MW_Float( WORD_STRONG:= MesBlock[1][1], 	WORD_WEAK := MesBlock[1][2],  VAR_OUT:=MesDataExd.MesData.MesI1);
MW_Float( WORD_STRONG:= MesBlock[1][3], 	WORD_WEAK := MesBlock[1][4],  VAR_OUT:=MesDataExd.MesData.MesI2);
MW_Float( WORD_STRONG:= MesBlock[1][5], 	WORD_WEAK := MesBlock[1][6],  VAR_OUT:=MesDataExd.MesData.MesI3);
MW_Float( WORD_STRONG:= MesBlock[1][7], 	WORD_WEAK := MesBlock[1][8],  VAR_OUT:=MesDataExd.MesData.MesI0);
MW_Float( WORD_STRONG:= MesBlock[1][15], 	WORD_WEAK := MesBlock[1][16], VAR_OUT:=MesDataExd.Thermal_Overload);
MW_Float( WORD_STRONG:= MesBlock[1][17], 	WORD_WEAK := MesBlock[1][18], VAR_OUT:=MesDataExd.MesData.MesFreq);


MesDataExd.Comut 			:= WORD_TO_BOOL(MesBlock[2][7]);
MesDataExd.CB_Close 		:= WORD_TO_BOOL(MesBlock[2][8]);
MesDataExd.CB_In_Alarm 		:= WORD_TO_BOOL(MesBlock[2][9]);
MesDataExd.Trip_Counter 	:= WORD_TO_INT(MesBlock[3][3]);

END_IF
END_METHOD

END_FUNCTION_BLOCK

// ---- 01_Equipement_Library/ProtectRelay/FB_ProtectRelay_REF615.TcPOU
FUNCTION_BLOCK FB_ProtectRelay_REF615 EXTENDS FB_ProtectRelay_Base
VAR_INPUT PERSISTENT
	{attribute 'OPC.UA.DA' := '1'} 
		ParamIPAddress				: STRING 	:= '192.168.20.66'; 	// (NA)Config: IP Adress of PV INverter
	{attribute 'OPC.UA.DA' := '1'} 
		ParamUnitID 				: BYTE  	:= 1; 			  		// (NA)   Modbus Unit ID. 
	{attribute 'OPC.UA.DA' := '1'} 
		ParamTCPPort				: UINT		:= 502;					// (NA) TCP port for modbus
		

//		ParamTempoComAlarm			: TIME 		:= T#2S;
//		ParamTempoComWarning		: TIME		:= T#2S;
		ParamNominalCurrent			: REAL 		:= 100 ; 				// (A) Nominal current set in the protection relay.
		
END_VAR

VAR
	// M_ALARMMANAGEMENT		
//		TON_ComAlarm				: TON;
//		TON_ComWarning				: TON;	
//		MesWarningCom				: BOOL;
//		MesAlarmCom					: BOOL;
	// M_READ VARIABLES//
		AX_ModbusRead		   		: ARRAY [1..3] OF FB_ModbusRead ; 					// (NA) FB for Modbus Reading
		                                        
		MesBlock_Temp 				: ARRAY [1..3] OF ARRAY[1..120]  OF WORD; 			// (NA) Temporary Block with multiple modbus reading (Caution : Double Word variables)

	MesDataExd		AT %Q* 	: ProtectRelay_REFIO ; 
	

	// M_STATEMANAGER//
	
END_VAR

METHOD M_AlarmManagement
//////////////////
// Manages IntelliGen Alarms
/////////////////

VAR 
	// Method local variables (reinitialized at each cycle) 
	FB_AlarmCodeManager : FB_AlarmCodeManager ; 

	KK					: BYTE;		// For Loop 
	
	ComWarning			: BOOL;		// Aggregated Wcommunication warning
	ComAlarm			: BOOL;		// Aggregated communication Alarm

	MesWarningCom: BOOL;
END_VAR

	//Alarm
	
	TON_ComAlarm	(IN:= (AX_ModbusRead[1].ModbusReadAlarm) AND (AX_ModbusRead[2].ModbusReadAlarm) AND (AX_ModbusRead[3].ModbusReadAlarm) , PT:= ParamTempoComAlarm, 	Q=> MesDataExd.MesData.MesAlarmCom) ;	
//	TON_ComWarning	(IN:= (AX_ModbusRead[1].ModbusReadAlarm) OR  (AX_ModbusRead[2].ModbusReadAlarm) OR  (AX_ModbusRead[3].ModbusReadAlarm) , PT:= ParamTempoComWarning, 	Q=>MesWarningCom) ;	

	MesWarningCom :=(AX_ModbusRead[1].ModbusReadAlarm) OR  (AX_ModbusRead[2].ModbusReadAlarm) OR  (AX_ModbusRead[3].ModbusReadAlarm) ; 


	
// ALARM CODE //
	FB_AlarmCodeManager(
		bAlarm1			:= MesDataExd.MesData.MesAlarmImax,  				//  Max I>>0  fault  
		bAlarm2			:= FALSE , 										//
		bAlarm3			:= MesDataExd.MesData.MesAlarmCom , 			// Communication alarm #COM
		bAlarm4			:= MesDataExd.MesData.MesAlarmTCS, 		        // Trip circuit Supervision alarm .     
		bAlarm5			:= FALSE, 										// 
		bAlarm6			:= FALSE, 										// 
		bAlarm7			:= False, 										// 
		bAlarm8			:= False, 										// 
		bAlarm9			:= FALSE, 										//
		bAlarm10		:= FALSE, 										//
		bAlarm11		:= FALSE,                       				//
		bAlarm12		:= FALSE,                       				//
		bAlarm13		:= FALSE, 										//
		bAlarm14		:= FALSE, 										// 
		bAlarm15		:= FALSE , 										// 
		wAlarmCode		=>MesDataExd.MesData.MesAlarmCode);

// WARNING CODE //
	FB_AlarmCodeManager(
 		bAlarm1			:= MesWarningCom,								// Bad communication	#COM			
		bAlarm2			:= FALSE ,										// 
		bAlarm3			:= FALSE , 										//		
		bAlarm4			:= FALSE, 						                //
		bAlarm5			:= FALSE, 						                //
		bAlarm6			:= FALSE, 						                //
		bAlarm7			:= FALSE,                                       //
		bAlarm8			:= FALSE,                                       //
		bAlarm9			:= FALSE,                                       //
		bAlarm10		:= FALSE,                                       //
		bAlarm11		:= FALSE,                                       //
		bAlarm12		:= FALSE,                                       //
		bAlarm13		:= FALSE,                                       //
		bAlarm14		:= FALSE,                                       //
		bAlarm15		:= FALSE,                                       //
		wAlarmCode		=>MesDataExd.MesData.MesWarningCode);	

// EVENT CODE //
	FB_AlarmCodeManager(
 		bAlarm1			:= FALSE,		//				
		bAlarm2			:= FALSE,	    //
		bAlarm3			:= FALSE,		//	
		bAlarm4			:= FALSE, 		//				
		bAlarm5			:= FALSE, 		//				
		bAlarm6			:= FALSE, 		//				
		bAlarm7			:= FALSE,       //
		bAlarm8			:= FALSE,       //
		bAlarm9			:= FALSE,       //
		bAlarm10		:= FALSE,       //
		bAlarm11		:= FALSE,       //
		bAlarm12		:= FALSE,       //
		bAlarm13		:= FALSE,       //
		bAlarm14		:= FALSE,       //
		bAlarm15		:= FALSE,       //
		wAlarmCode		=>MesDataExd.MesData.MesEventCode);
END_METHOD

METHOD M_Read
//////////////////
//  Read Modbus Variable for PCS . 
/////////////////
VAR 
	// Method local variables (reinitialized at each cycle) 
		
		AX_Addr				: ARRAY[1..3] OF UINT := [138, 		9409, 	171 ];
		AX_Qty				: ARRAY[1..3] OF UINT := [4, 		4, 	36	];
		
	
END_VAR
// CP-Read / Write 

MesDataExd.MesData.MesCP_Read := MesCP_Read ; 


// System BMS 
IF MesCP_Read  THEN	

AX_ModbusRead[1]
(
	pDestAddr 		:= ADR(MesBlock_Temp[1]),
	sIPAddr 		:= ParamIPAddress,
	tTimeout 		:= ParamTimeout,
	nQuantity 		:= AX_Qty[1],
	ntcpport 		:= ParamTCPPort,
	nMBAddr 		:= AX_Addr[1]-1,
	nUnitID 		:= ParamUnitID,
	cbLength 		:= SIZEOF(MesBlock_Temp[1]),
	ClockRead 		:= ClockRead AND MesCP_Read,
	Reset 			:= CmdClearFault_G OR IN_CmdReset_L,
);

AX_ModbusRead[2]
(
	pDestAddr 		:= ADR(MesBlock_Temp[2]),
	sIPAddr 		:= ParamIPAddress,
	tTimeout 		:= ParamTimeout,
	nQuantity 		:= AX_Qty[2],
	ntcpport 		:= ParamTCPPort,
	nMBAddr 		:= AX_Addr[2]-1,
	nUnitID 		:= ParamUnitID,
	cbLength 		:= SIZEOF(MesBlock_Temp[2]),
	ClockRead 		:= ClockRead AND MesCP_Read,
	Reset 			:= CmdClearFault_G OR IN_CmdReset_L
);

AX_ModbusRead[3]
(
	pDestAddr 		:= ADR(MesBlock_Temp[3]),
	sIPAddr 		:= ParamIPAddress,
	tTimeout 		:= ParamTimeout,
	nQuantity 		:= AX_Qty[3],
	ntcpport 		:= ParamTCPPort,
	nMBAddr 		:= AX_Addr[3]-1,
	nUnitID 		:= ParamUnitID,
	cbLength 		:= SIZEOF(MesBlock_Temp[3]),
	ClockRead 		:= ClockRead AND MesCP_Read,
	Reset 			:= CmdClearFault_G OR IN_CmdReset_L
);



	


MesDataExd.MesData.MesI1 	:= WORD_TO_REAL(MesBlock_Temp[1][1])/1000*ParamNominalCurrent;
MesDataExd.MesData.MesI2 	:= WORD_TO_REAL(MesBlock_Temp[1][2])/1000*ParamNominalCurrent;
MesDataExd.MesData.MesI3 	:= WORD_TO_REAL(MesBlock_Temp[1][3])/1000*ParamNominalCurrent;
MesDataExd.MesData.MesI0 	:= WORD_TO_REAL(MesBlock_Temp[1][4])/1000*ParamNominalCurrent;


MesDataExd.MesData.MesImax1	:= WORD_TO_REAL(MesBlock_Temp[2][1])/1000*ParamNominalCurrent;
MesDataExd.MesData.MesImax2	:= WORD_TO_REAL(MesBlock_Temp[2][2])/1000*ParamNominalCurrent;
MesDataExd.MesData.MesImax3	:= WORD_TO_REAL(MesBlock_Temp[2][3])/1000*ParamNominalCurrent;
MesDataExd.MesData.MesImax0	:= WORD_TO_REAL(MesBlock_Temp[2][4])/1000*ParamNominalCurrent;


MesDataExd.MesTransfoAlarm		:= MesBlock_Temp[3][31].0 ;
MesDataExd.MesSWOpened			:= MesBlock_Temp[3][31].4 ;
MesDataExd.MesSWClosed			:= MesBlock_Temp[3][31].6 ;
MesDataExd.MesEarth				:= MesBlock_Temp[3][31].8 ;
MesDataExd.MesSF6Low			:= MesBlock_Temp[3][31].10;
MesDataExd.MesSF6Unsufficient	:= MesBlock_Temp[3][31].12;
MesDataExd.MesTransfoWarning		:= MesBlock_Temp[3][31].14;

MesDataExd.MesClosed	        := MesBlock_Temp[3][30].2;
MesDataExd.MesOpened	        := MesBlock_Temp[3][30].4;
MesDataExd.MesComutLocal				:= NOT MesBlock_Temp[3][30].6;

MesDataExd.MesData.MesAlarmImax				:= MesBlock_Temp[3][3].1 ; // Max I ou Max I Inverse. Maintenu jusque l'acquittement.  
//MesDataExd.MesData.MesAlarmTCS				:=  ; 

END_IF

//MesDataExd.MesData.MesAlarmUminrmUmin	:= ; 

// Properties update
MesDataExd.MesData.MesI := (MesDataExd.MesData.MesI1 + MesDataExd.MesData.MesI2 + MesDataExd.MesData.MesI3)/3 ;
END_METHOD

END_FUNCTION_BLOCK

// ---- 01_Equipement_Library/ProtectRelay/FB_ProtectRelay_SepamT20.TcPOU
FUNCTION_BLOCK FB_ProtectRelay_SepamT20 EXTENDS FB_ProtectRelay_Base
//////////////////
// SEPAM system for High Voltage or Low Voltage Grid Protection . 
//////////////////
VAR_INPUT PERSISTENT
	// Parameters of the Object (instance/model specific) 
	 
END_VAR

VAR_OUTPUT
	//Child objects
	OutFBCompleteted						: BOOL;
END_VAR

VAR_INPUT
	InUnitID            : DINT;			// (NA)   ID FOR SEPAM T20 Modbus Unit ID. 

	// I/O Inputs		
END_VAR

VAR
	//M_Read
	FB_ModbusRead_I1						: FB_ReadModbusRTU_V2; 				// (NA) FB for Modbus Reading
	FB_ModbusRead_I2						: FB_ReadModbusRTU_V2; 				// (NA) FB for Modbus Reading
	FB_ModbusRead_I3						: FB_ReadModbusRTU_V2; 				// (NA) FB for Modbus Reading
	ParamTimeoutRTU							: TIME:=T#10S;
	MesBlock1_Temp							: ARRAY [0..36] OF WORD;
	MesBlock2_Temp							: WORD;
	MesBlock3_Temp							: WORD;
	MesModbusAlarmCode						: UDINT;							// (NA) Modbus Read Alarm Code
	MesModbusAlarmCode2						: UDINT;							// (NA) Modbus Read Alarm Code
	MesModbusAlarmCode3						: UDINT;							// (NA) Modbus Read Alarm Code
	ModbusReadAlarm 						: BOOL;								// (NA) Modbus Read Alarm for communications
	ModbusReadAlarm2 						: BOOL;	
	ModbusReadAlarm3 						: BOOL;	
	AX_bRead 								: ARRAY [1..3] OF BOOL;
	CalAllCompleted							: BOOL;
	//M_ALARMMANAGEMENT VARIABLES//

	//M_Execute
	AllNotBusy								: BOOL;
	TP_Read									: TP;
	RTrig									: R_TRIG;
//	ClockRead								: BOOL;
	
	//EValuate//
MesDataExd					AT %Q* 		: ProtectRelay_T20;
	

		
END_VAR

METHOD M_AlarmManagement
//////////////////
// Manages Sepam Alarms. Alarms opens HT CB until Sepam manual Reset . Warning Opens CB-L but does not maintain warning
/////////////////

VAR 
	// Method local variables (reinitialized at each cycle) 
	FB_AlarmCodeManager 	: FB_AlarmCodeManager ; 
 	ComWarning				: BOOL;
	ComAlarms				: BOOL;
END_VAR
ComWarning	:= ModbusReadAlarm OR ModbusReadAlarm2 OR ModbusReadAlarm3;
ComAlarms	:= ModbusReadAlarm OR ModbusReadAlarm2 OR ModbusReadAlarm3;

// ALARM CODE //
	FB_AlarmCodeManager(
		bAlarm1				:= FALSE,									//	
		bAlarm2				:= MesDataExd.MesGlobalWarming > 95 ,		// Calc of Warming TR from Sepam > 95 % OF T° Max				
		bAlarm3				:= ComAlarms ,								// Communication alarm  #COM
		bAlarm4				:= FALSE,     							//
		bAlarm5				:= FALSE,         						// 
		bAlarm6				:= FALSE, 								// 
		bAlarm7				:= FALSE, //
		bAlarm8				:= FALSE, //
		bAlarm9				:= FALSE, //
		bAlarm10			:= FALSE, //
		bAlarm11			:= FALSE, //
		bAlarm12			:= FALSE, //
		bAlarm13			:= FALSE, //
		bAlarm14			:= FALSE, //
		bAlarm15			:= FALSE , 	// 
		wAlarmCode			=>MesDataExd.MesData.MesAlarmCode);

// WARNING CODE //
	FB_AlarmCodeManager(
		bAlarm1			:= ComWarning, 							//  At least One Register do not responce #COM
		bAlarm2			:= FALSE,//  MesDataExd.MesData.MesPartialdefault, 			// Sepam in partial defaut IO, Tor fault
		bAlarm4			:= MesDataExd.MesGlobalWarming > 80, 	// Calc of Warming TR from Sepam > 80 % OF T° Max
		bAlarm5			:= FALSE, //
		bAlarm6			:= FALSE, //
		bAlarm7			:= FALSE, //
		bAlarm8			:= FALSE, //
		bAlarm9			:= FALSE, //
		bAlarm10		:= FALSE, //
		bAlarm11		:= FALSE, //
		bAlarm12		:= FALSE, //
		bAlarm13		:= FALSE, //
		bAlarm14		:= FALSE, //
		bAlarm15		:= FALSE, //
		wAlarmCode		=>MesDataExd.MesData.MesWarningCode);

// EVENT CODE //
	FB_AlarmCodeManager(
		bAlarm1			:=FALSE, 		// 
		bAlarm2			:=FALSE, 		// 
		bAlarm3			:=FALSE, 		// 
		bAlarm4			:=FALSE, 		// 
		bAlarm5			:=FALSE, 
		bAlarm6			:=FALSE, 
		bAlarm7			:=FALSE, 
		bAlarm8			:=FALSE, 
		bAlarm9			:=FALSE, 
		bAlarm10		:=FALSE, 
		bAlarm11		:=FALSE, 
		bAlarm12		:=FALSE, 
		bAlarm13		:=FALSE, 
		bAlarm14		:=FALSE, 
		bAlarm15		:=FALSE, 
		wAlarmCode		=>MesDataExd.MesData.MesEventCode);
END_METHOD

METHOD M_Init
VAR_INPUT
END_VAR
OutFBCompleteted := FALSE;
TP_Read(PT := ParamClockReadTime);
FB_ModbusRead_I1(InTimeout:= ParamTimeoutRTU,
				 InUnitID:= DINT_TO_BYTE(InUnitID),
				 InQuantity:= 36,	
				 InFunctionRead := 1);
				 
FB_ModbusRead_I2(InTimeout:= ParamTimeoutRTU,
				 InUnitID:= DINT_TO_BYTE(InUnitID),
				 InQuantity:= 1,	
				 InFunctionRead := 1);

				 
FB_ModbusRead_I3(InTimeout:= ParamTimeoutRTU,
				 InUnitID:= DINT_TO_BYTE(InUnitID),
				 InQuantity:= 1,	
				 InFunctionRead := 1);
END_METHOD

METHOD M_Read
//////////////////
//  Method Calls 
/////////////////

VAR 
//local variables (reinitialized at each cycle) 
	Busy1 : BOOL;
	Error1: BOOL;
	Busy2 : BOOL;
	Error2: BOOL;
	Busy3 : BOOL;
	Error3: BOOL;
	MW 					: FB_MergeWordsToDint; 
END_VAR
// CP-Read / Write 

MesDataExd.MesData.MesCP_Read := MesCP_Read ; 

IF MesCP_Read  THEN	



AllNotBusy:=TRUE;
AllNotBusy:=NOT(FB_ModbusRead_I1.OutBusy) AND NOT(FB_ModbusRead_I2.OutBusy) AND NOT(FB_ModbusRead_I3.OutBusy) AND AllNotBusy;



OutFBCompleteted:=FALSE;

// MODBUS REQUEST//
	//First register
		FB_ModbusRead_I1(InClockRead:= ClockRead,				
						InStartAddr:= 16#106,
						InAddrDest := ADR(MesBlock1_Temp),
						OutBusy => Busy1,
						OutErrorMbRead => Error1, 
						OutErrorId => MesModbusAlarmCode
						   );
						
		IF FB_ModbusRead_I1.OutbCompleted THEN
			ModbusReadAlarm := Error1;
			AX_bRead[1] 		:= TRUE;
		ELSIF NOT busy1 AND Error1 THEN
			ModbusReadAlarm := Error1;
		END_IF
	//Seconde Register
		FB_ModbusRead_I2(InClockRead:= ClockRead,				
						InStartAddr:= 16#1004,
						InAddrDest := ADR(MesBlock2_Temp),
						OutBusy => Busy2,
						OutErrorMbRead => Error2, 
						OutErrorId => MesModbusAlarmCode2
						   );		
		IF FB_ModbusRead_I2.OutbCompleted THEN
			ModbusReadAlarm2 := Error2;
			AX_bRead[2] 		:= TRUE;
		ELSIF NOT busy1 AND Error1 THEN
			ModbusReadAlarm2 := Error2;
		END_IF
	
	
	
	//Third Register
		FB_ModbusRead_I3(InClockRead:= ClockRead,				
						InStartAddr:= 16#1007,
						InAddrDest := ADR(MesBlock3_Temp),
						OutBusy => Busy3,
						OutErrorMbRead => Error3, 
						OutErrorId => MesModbusAlarmCode3
						   );		
		IF FB_ModbusRead_I3.OutbCompleted THEN
			ModbusReadAlarm3 := Error3;
			AX_bRead[3] 		:= TRUE;
		ELSIF NOT busy3 AND Error3 THEN
			ModbusReadAlarm3 := Error3;
		END_IF
	
	
CalAllCompleted :=  AX_bRead[1] AND AX_bRead[2] AND AX_bRead[3];
OutFBCompleteted := CalAllCompleted;	

//CHECK IF ALL MODBUS REQUESTS ARE FINISHED
	IF (CalAllCompleted) THEN
//RESETING CLOCK READ FOR EACH REQUEST
		AX_bRead[1]:= FALSE;
		AX_bRead[2]:= FALSE;
		AX_bRead[3]:= FALSE;
		CalAllCompleted := FALSE;
	END_IF
	
MW( WORD_STRONG:= MesBlock1_Temp[0], SIGNED:=FALSE, FIX:=0 , SIZE:=1, VAR_OUT 	:=MesDataExd.MesData.MesI1);
MW( WORD_STRONG:= MesBlock1_Temp[1], SIGNED:=FALSE, FIX:=0 , SIZE:=1, VAR_OUT 	:=MesDataExd.MesData.MesI2);
MW( WORD_STRONG:= MesBlock1_Temp[2], SIGNED:=FALSE, FIX:=0 , SIZE:=1, VAR_OUT 	:=MesDataExd.MesData.MesI3);
MW( WORD_STRONG:= MesBlock1_Temp[33], SIGNED:=FALSE, FIX:=2 , SIZE:=1, VAR_OUT	:=MesDataExd.MesData.MesFreq);
MW( WORD_STRONG:= MesBlock1_Temp[34], SIGNED:=TRUE, FIX:=0 , SIZE:=1, VAR_OUT 	:=MesDataExd.MesP);
MW( WORD_STRONG:= MesBlock1_Temp[35], SIGNED:=TRUE, FIX:=0 , SIZE:=1, VAR_OUT 	:=MesDataExd.MesQ);
MW( WORD_STRONG:= MesBlock1_Temp[36], SIGNED:=TRUE, FIX:=0 , SIZE:=1, VAR_OUT 	:=MesDataExd.MesS);
MW( WORD_STRONG:= MesBlock2_Temp, SIGNED:=FALSE, FIX:=-1 , SIZE:=1, VAR_OUT 	:=MesDataExd.MesTripProtec);
MW( WORD_STRONG:= MesBlock3_Temp, SIGNED:=FALSE, FIX:=0 , SIZE:=1, VAR_OUT 		:=MesDataExd.MesGlobalWarming);

END_IF
END_METHOD

END_FUNCTION_BLOCK

// ---- 01_Equipement_Library/ProtectRelay/FB_ProtectRelay_VIP410.TcPOU
FUNCTION_BLOCK FB_ProtectRelay_VIP410 EXTENDS FB_ProtectRelay_Base
//////////////////
// SEPAM system for High Voltage or Low Voltage Grid Protection . 
//////////////////
VAR_INPUT PERSISTENT
	{attribute 'OPC.UA.DA' := '1'} 
	ParamTcpPort				: UINT:=502;		(* (NA) Tcp port *)
	{attribute 'OPC.UA.DA' := '1'} 
	ParamIPAddress				: STRING;       	(* (NA) IP address*)
	{attribute 'OPC.UA.DA' := '1'} 
	ParamUnitID					: BYTE;         	(* (NA) Unit ID*)
	{attribute 'OPC.UA.DA' := '1'}
	ParamClockInputTime 		: TIME:= TIME#5S;   (* (Time) Read Modbus Frequency*)
END_VAR

VAR_OUTPUT
	
END_VAR

VAR_INPUT
	IN_MesTrip_IO				: BOOL ; 
END_VAR

VAR
	
	MesDataExd		AT %Q* 		: ProtectRelay_VIP410;
	FB_ModbusRead	          	: ARRAY[1..4] OF FB_ModbusRead; 
	ClockReadInput				: BOOL;

	MesBlock1_Temp 				: ARRAY [1..1] OF WORD ; 
	MesBlock2_Temp 				: ARRAY [1..20] OF WORD ; 
	MesBlock3_Temp 				: ARRAY [1..8] OF WORD ; 
	MesBlock4_Temp 				: ARRAY [1..2] OF WORD ; 
	AX_ModbusReadAlarm			: ARRAY[1..4] OF BOOL;
	AX_ModbusReadAlarmId		: ARRAY[1..4] OF UDINT;	
END_VAR

METHOD M_AlarmManagement
//////////////////
// Manages Sepam Alarms. Alarms opens HT CB until Sepam manual Reset . Warning Opens CB-L but does not maintain warning
/////////////////

VAR 
	// Method local variables (reinitialized at each cycle) 
	FB_AlarmCodeManager 	: FB_AlarmCodeManager ; 
	RS_Trip					: SR;
	ComWarning: BOOL ;
END_VAR
RS_Trip(SET1 := IN_MesTrip_IO  , Reset := CmdClearFault_G OR IN_CmdReset_L ); // SR FB for keep fire if burn .

TON_ComAlarm(IN:= AX_ModbusReadAlarm[1] AND AX_ModbusReadAlarm[2] AND AX_ModbusReadAlarm[3] AND AX_ModbusReadAlarm[4] , PT:= ParamTempoComAlarm, Q=>MesdataExd.MesData.MesAlarmCom) ;	

ComWarning := AX_ModbusReadAlarm[1] OR AX_ModbusReadAlarm[2] OR AX_ModbusReadAlarm[3] OR AX_ModbusReadAlarm[4] ; 

// ALARM CODE //
	FB_AlarmCodeManager(
		bAlarm1				:= RS_Trip.Q1,							// General trip
		bAlarm2				:= NOT IN_MesWatchDog_IO,				// Watchdog lost
		bAlarm3				:= MesdataExd.MesData.MesAlarmCom,		// Communication Alarm
		bAlarm4				:= FALSE,     							// 
		bAlarm5				:= FALSE,         						// 
		bAlarm6				:= FALSE, 								// 
		bAlarm7				:= FALSE, 								// 
		bAlarm8				:= FALSE, 								// 
		bAlarm9				:= FALSE, 								// 
		bAlarm10			:= FALSE, 								// 
		bAlarm11			:= FALSE, 								// 
		bAlarm12			:= FALSE, 								// 
		bAlarm13			:= FALSE, 								// 
		bAlarm14			:= FALSE, 								// 
		bAlarm15			:= FALSE,								//  	
		wAlarmCode			=> MesdataExd.MesData.MesAlarmCode);

// WARNING CODE //
	FB_AlarmCodeManager(
		bAlarm1			:= FALSE,									// 
		bAlarm2			:= FALSE,									// 
		bAlarm4			:= FALSE,									// 
		bAlarm5			:= FALSE,									// 
		bAlarm6			:= FALSE,									// 
		bAlarm7			:= FALSE,									//  
		bAlarm8			:= FALSE,									// 
		bAlarm9			:= FALSE,									// 
		bAlarm10		:= FALSE,									// 
		bAlarm11		:= FALSE,									// 
		bAlarm12		:= FALSE,									// 
		bAlarm13		:= FALSE,									// 
		bAlarm14		:= FALSE,									//
		bAlarm15		:= FALSE,									//
		wAlarmCode		=> MesdataExd.MesData.MesWarningCode);

// EVENT CODE //
	FB_AlarmCodeManager(
		bAlarm1			:=FALSE, 									// 
		bAlarm2			:=FALSE, 									// 
		bAlarm3			:=FALSE, 									// 
		bAlarm4			:=FALSE, 									// 
		bAlarm5			:=FALSE, 									// 
		bAlarm6			:=FALSE, 									// 
		bAlarm7			:=FALSE, 									// 
		bAlarm8			:=FALSE, 									// 
		bAlarm9			:=FALSE, 									// 
		bAlarm10		:=FALSE, 									// 
		bAlarm11		:=FALSE, 									// 
		bAlarm12		:=FALSE, 									// 
		bAlarm13		:=FALSE, 									// 
		bAlarm14		:=FALSE, 									//
		bAlarm15		:=FALSE, 									//
		wAlarmCode		=> MesdataExd.MesData.MesEventCode);
END_METHOD

METHOD M_Evaluate
VAR_INPUT
END_VAR

VAR
END_VAR

// Structure update 
	MesDataExd.MesData.MesI		:= (MesDataExd.MesData.MesI1 + MesDataExd.MesData.MesI2 + MesDataExd.MesData.MesI3 )/3 ; 
	///MesDataExd.MesData	:= MesData;
END_METHOD

METHOD M_Init
VAR_INPUT
END_VAR
END_METHOD

METHOD M_Read
//////////////////
//  Method Calls 
/////////////////

VAR_INPUT
	
END_VAR
VAR 
	MW					: FB_MergeWordsToFloat;
END_VAR
// CP-Read / Write 

MesDataExd.MesData.MesCP_Read := MesCP_Read ; 

IF MesCP_Read  THEN	



FB_ModbusRead[1]
	(
		nTCPPort		:= ParamTcpPort,
		ClockRead		:= MesCP_Read AND ClockRead	, 
		Reset			:= CmdClearFault_G OR IN_CmdReset_L,
		sIPAddr			:= ParamIPAddress ,
		nUnitID			:= ParamUnitID, 
		tTimeout		:= T#5S,
		nQuantity		:= 1, 
		nMBAddr			:= 40000 , 
		cbLength		:= SIZEOF(MesBlock1_Temp) , 
		pDestAddr		:= ADR(MesBlock1_Temp) , 
		ModbusReadAlarm	=> AX_ModbusReadAlarm[1] , 
		ErrorId			=> AX_ModbusReadAlarmId[1]
	);
	
FB_ModbusRead[2]
	(
		nTCPPort		:= ParamTcpPort,
		ClockRead		:= MesCP_Read AND ClockRead	, 
		Reset			:= CmdClearFault_G OR IN_CmdReset_L,
		sIPAddr			:= ParamIPAddress ,
		nUnitID			:= ParamUnitID, 
		tTimeout		:= T#5S,
		nQuantity		:= 20, 
		nMBAddr			:= 40200 , 
		cbLength		:= SIZEOF(MesBlock2_Temp) , 
		pDestAddr		:= ADR(MesBlock2_Temp) , 
		ModbusReadAlarm	=> AX_ModbusReadAlarm[2], 
		ErrorId			=> AX_ModbusReadAlarmId[2]
	);

FB_ModbusRead[3]
	(
		nTCPPort		:= ParamTcpPort,
		ClockRead		:= MesCP_Read AND ClockRead	, 
		Reset			:= CmdClearFault_G OR IN_CmdReset_L,
		sIPAddr			:= ParamIPAddress ,
		nUnitID			:= ParamUnitID, 
		tTimeout		:= T#5S,
		nQuantity		:= 8, 
		nMBAddr			:= 40254 , 
		cbLength		:= SIZEOF(MesBlock3_Temp) , 
		pDestAddr		:= ADR(MesBlock3_Temp) , 
		ModbusReadAlarm	=> AX_ModbusReadAlarm[3], 
		ErrorId			=> AX_ModbusReadAlarmId[3]
	);
	
FB_ModbusRead[4]
	(
		nTCPPort		:= ParamTcpPort,
		ClockRead		:= MesCP_Read AND ClockRead	, 
		Reset			:= CmdClearFault_G OR IN_CmdReset_L,
		sIPAddr			:= ParamIPAddress ,
		nUnitID			:= ParamUnitID, 
		tTimeout		:= T#5S,
		nQuantity		:= 2, 
		nMBAddr			:= 40351 , 
		cbLength		:= SIZEOF(MesBlock4_Temp) , 
		pDestAddr		:= ADR(MesBlock4_Temp) , 
		ModbusReadAlarm	=> AX_ModbusReadAlarm[4], 
		ErrorId			=> AX_ModbusReadAlarmId[4]
	);
	
	//COM
	MesdataExd.MesStatCom := WORD_TO_BOOL(MesBlock1_Temp[1]);
	//I
	MW( WORD_STRONG:= MesBlock2_Temp[2  ],	WORD_WEAK := MesBlock2_Temp[1  ], VAR_OUT := MesDataExd.MesData.MesI1 );		
	MW( WORD_STRONG:= MesBlock2_Temp[4  ],	WORD_WEAK := MesBlock2_Temp[3  ], VAR_OUT := MesDataExd.MesData.MesI2 );	
	MW( WORD_STRONG:= MesBlock2_Temp[6  ],	WORD_WEAK := MesBlock2_Temp[5  ], VAR_OUT := MesDataExd.MesData.MesI3 );
	MW( WORD_STRONG:= MesBlock2_Temp[8  ],	WORD_WEAK := MesBlock2_Temp[7  ], VAR_OUT := MesDataExd.MesData.MesI0 );	
	
	//AvgI
	MW( WORD_STRONG:= MesBlock2_Temp[10  ],	WORD_WEAK := MesBlock2_Temp[9  ], VAR_OUT 	:= MesDataExd.MesAvgI1 );	
	MW( WORD_STRONG:= MesBlock2_Temp[12  ],	WORD_WEAK := MesBlock2_Temp[11  ], VAR_OUT 	:= MesDataExd.MesAvgI2 );	
	MW( WORD_STRONG:= MesBlock2_Temp[14  ],	WORD_WEAK := MesBlock2_Temp[13  ], VAR_OUT 	:= MesDataExd.MesAvgI3 );	
	//Imax
	MW( WORD_STRONG:= MesBlock2_Temp[16  ],	WORD_WEAK := MesBlock2_Temp[15 ], VAR_OUT  := MesDataExd.MesData.MesImax1 );	
	MW( WORD_STRONG:= MesBlock2_Temp[18  ],	WORD_WEAK := MesBlock2_Temp[17  ], VAR_OUT := MesDataExd.MesData.MesImax2 );	
	MW( WORD_STRONG:= MesBlock2_Temp[20  ],	WORD_WEAK := MesBlock2_Temp[19  ], VAR_OUT := MesDataExd.MesData.MesImax3 );	

	//Itrip
	MW( WORD_STRONG:= MesBlock3_Temp[2  ],	WORD_WEAK := MesBlock3_Temp[1  ], VAR_OUT := MesDataExd.MesData.MesImax1 );		
	MW( WORD_STRONG:= MesBlock3_Temp[4  ],	WORD_WEAK := MesBlock3_Temp[3  ], VAR_OUT := MesDataExd.MesData.MesImax2 );	
	MW( WORD_STRONG:= MesBlock3_Temp[6  ],	WORD_WEAK := MesBlock3_Temp[5  ], VAR_OUT := MesDataExd.MesData.MesImax3 );
	MW( WORD_STRONG:= MesBlock3_Temp[8  ],	WORD_WEAK := MesBlock3_Temp[7  ], VAR_OUT := MesDataExd.MesI0Fault );	

	MesdataExd.ControlWord 	:= MesBlock4_Temp[1];
	MesdataExd.StatusWord 	:= MesBlock4_Temp[2];
	
END_IF
END_METHOD

END_FUNCTION_BLOCK

// ---- 01_Equipement_Library/ProtectRelay/FB_ProtectRelay_WIP1.TcPOU
FUNCTION_BLOCK FB_ProtectRelay_WIP1 EXTENDS FB_ProtectRelay_Base
VAR_INPUT
						
	
	

END_VAR

VAR_INPUT
	// I/O Inputs 		                                     				
		IN_MesAlarmImax_IO		: BOOL ; // IO max I  fault
		IN_MesAlarmUmin_IO		: BOOL ;  // IO Min U  Fault 
		
END_VAR


VAR
// M_ALARMMNGMT VARIABLES //
                            		
	CmdResetHVCell				: BOOL ; 
	// M_READ VARIABLES//
	
MesDataExd 		    AT %Q*  	: ProtectRelay_WIP1; 	
		


END_VAR

METHOD M_AlarmManagement
VAR 
	// Method local variables (reinitialized at each cycle) 
	FB_AlarmCodeManager : FB_AlarmCodeManager ; 

	ComWarning: BOOL;
	ComAlarm: BOOL;
	KK: BYTE;
	
END_VAR
// Detection Variables

MesDataExd.MesData.MesAlarmImax	:= IN_MesAlarmImax_IO ; 
MesDataExd.MesData.MesAlarmUmin :=  IN_MesAlarmUmin_IO ; 


// ALARM CODE //
	FB_AlarmCodeManager(
		bAlarm1	 := MesDataExd.MesData.MesAlarmImax,// Max I Fault 
		bAlarm2	 := MesDataExd.MesData.MesAlarmUmin,// Min U  Fault
		bAlarm3	 := FALSE, //
		bAlarm4	 := FALSE,//
		bAlarm5	 := FALSE, //
		bAlarm6	 := FALSE,//
		bAlarm7	 := FALSE, //
		bAlarm8	 := FALSE,//
		bAlarm9	 := FALSE, //
		bAlarm10 := FALSE,//
		bAlarm11 := FALSE, //
		bAlarm12 := FALSE,//
		bAlarm13 := FALSE, //
		bAlarm14 := FALSE,//														   
		bAlarm15 := FALSE,//									                      
		wAlarmCode	=>MesDataExd.MesData.MesAlarmCode);


// WARNING CODE //
	FB_AlarmCodeManager(
 		bAlarm1			:= FALSE, //
		bAlarm2			:= FALSE,//
        bAlarm3			:= FALSE, //
		bAlarm4			:= FALSE,// 
		bAlarm5			:= FALSE, // 
		bAlarm6			:= FALSE,// 
		bAlarm7			:= FALSE, // 
		bAlarm8			:= FALSE,// 
		bAlarm9			:= FALSE, // 
		bAlarm10		:= FALSE,// 
		bAlarm11		:= FALSE, // 
		bAlarm12		:= FALSE,//		 
		bAlarm13		:= FALSE,//		 
		bAlarm14		:= FALSE,  //
		bAlarm15		:= FALSE, //
		wAlarmCode	=>MesDataExd.MesData.MesWarningCode);
END_METHOD

METHOD M_Execute

// INITIALIZE // 
	IF bInit THEN
		M_Init() ; 
		bInit		:= FALSE ; 
		
	ELSIF IN_CmdReset_L THEN 
		bInit		:= TRUE ;
		
	END_IF





M_AlarmManagement() ;
END_METHOD

END_FUNCTION_BLOCK

// ---- 01_Equipement_Library/ProtectRelay/FB_ProtectRelay_SEPAM10a.TcPOU
FUNCTION_BLOCK FB_ProtectRelay_SEPAM10a EXTENDS FB_ProtectRelay_Base
VAR_INPUT
	InUnitID            : DINT;			// (NA)   SMA Modbus Unit ID. 
	
END_VAR
VAR_OUTPUT
	OutFBCompleteted   : BOOL;
	
END_VAR
VAR
// M_ALARMMNGMT VARIABLES //
		MesAlarmCode				: WORD ;  			// (NA) [P,H,B]   Alarm Word . 0: Synthesis , 1:SMA general alarm , 2:Communication Alarm , 3:, 4:, 5:, 6:, 7:, 8:, 9:, 10:, 11:, 12:, 13:, 14:, 15:, 16:
		MesWarningCode				: WORD ;  			// (NA) [P,H,B]   Warning Word . 0: Synthesis , 1:SMA general warning  , 2: , 3: , 4:, 5:, 6:, 7:, 8:, 9:, 10:, 11:, 12:, 13:, 14:, 15:, 16:		
  		MesEventCode				: WORD; 			// (NA) [P,H,B] Event Code. Acknowledgable.
                                              		

		MesComError					: BOOL ; 			// (NA) [P,H]  True if lost of communication
		MesAlarmCom					: BOOL ; 			// (NA) All modbus trame fail 
		
	// M_READ VARIABLES//
		FB_ModbusRead_I1          	: FB_ReadModbusRTU_V2; 				// (NA) FB for Modbus Reading
		MesDataExd		      	AT %Q* 	: ProtectRelay_S48; 	
		MesBlock1_Temp 				: ARRAY[0..7]  OF WORD; 			// (NA) Temporary Block with multiple modbus reading (Caution : Double Word variables)
		AX_bRead 					: ARRAY[1..2]  OF BOOL;
		ModbusReadAlarm             : BOOL;				// (NA) Modbus Read Alarm for communications
		MesModbusAlarmCode			: UDINT;							// (NA) Modbus Read Alarm Code
		CalAllCompleted				: BOOL;								// (NA) Returns the status of all modbus requests
	
		AllNotBusy					: BOOL:=TRUE;
		TP_Read						: LTP; 								// (NA) Tempo to define Modbus Reading Frequency
	//	ClockRead					: BOOL;								// (NA) Modbus reading Clock
		RTrig						: R_TRIG;
END_VAR

VAR CONSTANT
	    CstClockReadTime 		: LTIME := LTIME#1S;	  				// (Time) Read Modbus Frequency .	
END_VAR

METHOD M_AlarmManagement
VAR 
	// Method local variables (reinitialized at each cycle) 
	FB_AlarmCodeManager : FB_AlarmCodeManager ; 

	ComWarning: BOOL;
	ComAlarm: BOOL;
	KK: BYTE;
	
END_VAR
// Detection Variables
ComWarning 	:= ComWarning OR ModbusReadAlarm ; // At least one modbus trame did not work
ComAlarm	:= ComAlarm AND ModbusReadAlarm;  // All modbus trame did not work

MesComError := ComWarning ;  
MesAlarmCom := ComAlarm ;

// ALARM CODE //
	FB_AlarmCodeManager(
		bAlarm1	 := FALSE,//
		bAlarm2	 := FALSE,//
		bAlarm3	 := FALSE, 
		bAlarm4	 := FALSE,
		bAlarm5	 := FALSE,
		bAlarm6	 := FALSE,
		bAlarm7	 := FALSE,
		bAlarm8	 := FALSE,
		bAlarm9	 := FALSE,
		bAlarm10 := FALSE,
		bAlarm11 := FALSE,
		bAlarm12 := FALSE,
		bAlarm13 := FALSE,
		bAlarm14 := FALSE,														   
		bAlarm15 := FALSE,									                      
		wAlarmCode	=> MesAlarmCode);


// WARNING CODE //
	FB_AlarmCodeManager(
 		bAlarm1			:= FALSE,
		bAlarm2			:= FALSE,
        bAlarm3			:= FALSE,
		bAlarm4			:= FALSE, 
		bAlarm5			:= FALSE, 
		bAlarm6			:= FALSE, 
		bAlarm7			:= FALSE, 
		bAlarm8			:= FALSE, 
		bAlarm9			:= FALSE, 
		bAlarm10		:= FALSE, 
		bAlarm11		:= FALSE, 
		bAlarm12		:= FALSE, 
		bAlarm13		:= FALSE, 
		bAlarm14		:= FALSE, 
		bAlarm15		:= FALSE, 
		wAlarmCode	=> MesWarningCode);	
		
		
// EVENT CODE //
	FB_AlarmCodeManager(
		bAlarm1			:= FALSE,
		bAlarm2			:= FALSE,
		bAlarm3			:= FALSE,
		bAlarm4			:= FALSE, 		
		bAlarm5			:= FALSE, 
		bAlarm6			:= FALSE, 
		bAlarm7			:= FALSE, 
		bAlarm8			:= FALSE, 
		bAlarm9			:= FALSE, 
		bAlarm10		:= FALSE, 
		bAlarm11		:= FALSE, 
		bAlarm12		:= FALSE, 
		bAlarm13		:= FALSE, 
		bAlarm14		:= FALSE, 
		bAlarm15		:= FALSE, 
		wAlarmCode		=> MesEventCode);
END_METHOD

METHOD M_Execute
// INITIALIZE //
	IF NOT(bInit) THEN
		THIS^.M_Init();
		bInit := TRUE;
		
	END_IF
	IF bInit THEN
		AllNotBusy:=TRUE;
		AllNotBusy:=NOT(FB_ModbusRead_I1.OutBusy) AND AllNotBusy;
		TP_Read(In := NOT(TP_Read.Q) AND AllNotBusy);
		RTrig(CLK := TP_Read.Q);
		ClockRead := RTrig.Q;	
	// METHODS CALLS //
		// Order is important 
		THIS^.M_Read();
		THIS^.M_Evaluate();
	END_IF
END_METHOD

METHOD M_Init


VAR

END_VAR
OutFBCompleteted := FALSE;
TP_Read(PT := CstClockReadTime);

FB_ModbusRead_I1(
	InUnitID:= DINT_TO_BYTE(InUnitID), 
	InTimeout:= T#5s, 
	InFunctionRead:= 1 );
END_METHOD

METHOD M_Read

VAR
//local variables (reinitialized at each cycle) 
	Busy1 : BOOL;
	Error1: BOOL;
	
END_VAR
// CP-Read / Write 

MesDataExd.MesData.MesCP_Read := MesCP_Read ; 

IF MesCP_Read  THEN	
OutFBCompleteted:=FALSE;


// MODBUS REQUEST//
	FB_ModbusRead_I1(InClockRead:= ClockRead,				
					InStartAddr:= 16#113,
			   		InAddrDest := ADR(MesBlock1_Temp),
					OutBusy => Busy1,
					OutErrorMbRead => Error1, 
					OutErrorId => MesModbusAlarmCode
					   );
					
	IF FB_ModbusRead_I1.OutbCompleted THEN
		ModbusReadAlarm := Error1;
		AX_bRead[1] := TRUE;
	ELSIF NOT busy1 AND Error1 THEN
		ModbusReadAlarm := Error1;
		
	END_IF
	
	CalAllCompleted :=  AX_bRead[1];
	OutFBCompleteted := CalAllCompleted;
	
//CHECK IF ALL MODBUS REQUESTS ARE FINISHED
	IF (CalAllCompleted) THEN
//RESETING CLOCK READ FOR EACH REQUEST
		AX_bRead[1] := FALSE;
		CalAllCompleted := FALSE;
		
	END_IF
	
	
	
	//Block 1
	MesDataExd.MesData.MesI1  := (WORD_TO_INT(MesBlock1_Temp[1])/10);
MesDataExd.MesData.MesI2 := (WORD_TO_INT(MesBlock1_Temp[3])/10);
MesDataExd.MesData.MesI3 := (WORD_TO_INT(MesBlock1_Temp[5])/10);
	//MW(InFirstWord := MesBlock1_Temp[6],InSecondWord := MesBlock1_Temp[7],OutCalReal =>MesDataExd.MesData.MesRes_Ins);*)

END_IF
END_METHOD

END_FUNCTION_BLOCK

// ---- 01_Equipement_Library/ProtectRelay/FB_ProtectRelay_SepamS48.TcPOU
FUNCTION_BLOCK FB_ProtectRelay_SepamS48 EXTENDS FB_ProtectRelay_Base
//////////////////
// SEPAM system for High Voltage or Low Voltage Grid Protection. 
//////////////////

VAR_INPUT PERSISTENT
	// Parameters of the Object (instance/model specific) 
	   ParamTimeoutRTU						: TIME  := T#10S;					(* (s)	  Com RTU Timeout *)
	   ParamUnitID							: BYTE 	:= 1;						(* (NA)	  unit ID*)
	   ParamInInterfaceSub					: BOOL;								(* (NA)   Serial interface RS422/RS485 TYPE (0:EL6021, 1:SUB9)*)
END_VAR

VAR_OUTPUT
	//Child objects
	OUT_Protect_GTE_LONG_Running			: BOOL; 							// Long GTE fault, PP stop for 2m and lost of autorisation 

END_VAR

VAR_INPUT
	// I/O Inputs	
	IN_MesAlarmIMax_IO						: BOOL; 							// I max fault Fault, Losing autorisation and not possible to consumed
	IN_MesAlarmUmin_IO						: BOOL; 							// U min Fault, Keeping autorisation, If we have 3 gte in 30 min ==> Stop fedding and consumed during 2h
	IN_MesAlarmPWH_IO						: BOOL; 							// Defaut wattmétrique
	                                                								                                                	
	IN_CmdReset_3GTEFault					: BOOL; 							// 3GTE Fault Reset 
		
END_VAR

VAR
	//M_Read
	Trig_Read								: R_TRIG;
	ModbusRTU								: FB_ModbusRTU ;					// (NA) FB for Modbus Reading
	MbStruct								: ARRAY[1..2] OF Struct_InputRTU;

                                			
	ModbusAlarm								: ARRAY[1..2] OF BOOL;				// (NA) Read alarm
	AX_Quantity								: ARRAY[1..2] OF WORD;				// (NA) Quantity of blocks to read
	AX_Address								: ARRAY[1..2] OF WORD;				// (NA) Start address of the read
	OutErrorMbRead							: ARRAY[1..2] OF BOOL;
                                			
	Busy									: BOOL;
	MesBlock_Temp							: ARRAY [1..2] OF ARRAY [0..94] OF WORD;
	                            			
	RTrigI									: R_TRIG;
MesDataExd			AT %Q* 		: ProtectRelay_S48; 
	                            			
	//M_EVALUATE                			
	TON_GteIsLong							: TON;

	FB_3GTE									: FB_CountNinTimeWindow; 
	

END_VAR

METHOD M_AlarmManagement
//////////////////
// Manages Sepam Alarms. Alarms opens HT CB until Sepam manual reset. Warning opens CB-L but does not maintain warning.
/////////////////

VAR 
	// Method local variables (reinitialized at each cycle) 
	FB_AlarmCodeManager 	: FB_AlarmCodeManager ; 
 	ComWarning				: BOOL;
	ComAlarms				: BOOL;
END_VAR
ComWarning	:= OutErrorMbRead[1] OR OutErrorMbRead[2];
ComAlarms	:= OutErrorMbRead[1];

TON_ComAlarm(IN:= ComAlarms , PT:= ParamTempoComAlarm, Q=> MesDataExd.MesData.MesAlarmCom) ;	

// ALARM CODE //
	FB_AlarmCodeManager(
		bAlarm1				:= MesDataExd.MesData.MesAlarmUmin , 		// Min U Fault 
		bAlarm2				:= FALSE ,									//
		bAlarm3				:= NOT IN_MesWatchDog_IO,					// Watchdog TRUE := OK, False = Dead #COM
		bAlarm4				:= MesDataExd.MesData.MesAlarmImax,     	// C13100 Fault (Max I) 
		bAlarm5				:= FALSE,         							// 
		bAlarm6				:= FALSE, 									// 
		bAlarm7				:= FALSE, 									// 
		bAlarm8				:= FALSE, 									// 
		bAlarm9				:= FALSE, 									// 
		bAlarm10			:= FALSE, 									// 
		bAlarm11			:= FALSE, 									// 
		bAlarm12			:= FALSE, 									// 
		bAlarm13			:= FALSE, 									// 
		bAlarm14			:= FALSE, 									// 
		bAlarm15			:= FALSE ,									//  	
		wAlarmCode			=>MesDataExd.MesData.MesAlarmCode);

// WARNING CODE //
	FB_AlarmCodeManager(
		bAlarm1			:= ComWarning, 									// At least one register do not respond #COM
		bAlarm2			:= MesDataExd.MesData.MesAlarmCom ,				// Communication alarm #COM
		bAlarm3			:= FALSE , 										//		
		bAlarm4			:= FALSE , 										//
		bAlarm5			:= FALSE , 										//
		bAlarm6			:= IN_MesAlarmPWH_IO, 							// Wattmetric fault	
		bAlarm7			:= MesDataExd.MesData.MesAlarmUmin_Long, 		// Long Min U Fault (> 50s)
		bAlarm8			:= MesDataExd.MesData.MesAlarm_GTE3Time, 		// 3 min U fault in a row (GTE 3 times)
		bAlarm9			:= FALSE, 										//
		bAlarm10		:= FALSE, 										//
		bAlarm11		:= FALSE, 										//
		bAlarm12		:= FALSE, 										//
		bAlarm13		:= FALSE, 										//
		bAlarm14		:= FALSE, 										//
		bAlarm15		:= FALSE, 										//
		wAlarmCode		=>MesDataExd.MesData.MesWarningCode);

// EVENT CODE //
	FB_AlarmCodeManager(
		bAlarm1			:=FALSE, 										// 
		bAlarm2			:=FALSE, 										// 
		bAlarm3			:=FALSE, 										// 
		bAlarm4			:=FALSE, 										// 
		bAlarm5			:=FALSE, 										//
		bAlarm6			:=FALSE, 										//
		bAlarm7			:=FALSE, 										//
		bAlarm8			:=FALSE, 										//
		bAlarm9			:=FALSE, 										//
		bAlarm10		:=FALSE, 										//
		bAlarm11		:=FALSE, 										//
		bAlarm12		:=FALSE, 										//
		bAlarm13		:=FALSE, 										//
		bAlarm14		:=FALSE, 										//
		bAlarm15		:=FALSE, 										//
		wAlarmCode		=>MesDataExd.MesData.MesEventCode);
END_METHOD

METHOD M_Evaluate
VAR_INPUT
END_VAR

VAR

END_VAR
// GTE IS LONG AFTER 50S
TON_GteIsLong(IN:=IN_MesAlarmUmin_IO ,PT:=T#50S); 
MesDataExd.MesData.MesAlarmUmin_Long := TON_GteIsLong.Q ; 




FB_3GTE(IN_bInput := IN_MesAlarmUmin_IO , IN_bReset := IN_CmdReset_3GTEFault , IN_CountMax := 3 , ParamTimeToMeasure := T#30M , OUT_FlagNinT =>MesDataExd.MesData.MesAlarm_GTE3Time ) ; 
	



//Update MesData
MesDataExd.MesData.MesI			:= (MesDataExd.MesData.MesI1 + MesDataExd.MesData.MesI2 + MesDataExd.MesData.MesI3) / 3 ;
MesDataExd.MesData.MesAlarmUmin := IN_MesAlarmUmin_IO;
MesDataExd.MesData.MesAlarmImax	:= IN_MesAlarmIMax_IO;

MesDataExd.MesStopPP_UminLong 	:= OUT_Protect_GTE_LONG_Running;
END_METHOD

METHOD M_Init
VAR_INPUT
END_VAR
END_METHOD

METHOD M_Read
//////////////////
//  Method Calls 
/////////////////

VAR 
	MW 					: FB_MergeWordsToDint; 
	KK : UINT;

	AX_Addr					: ARRAY[1..2] OF UINT 	:= [16#113,		16#10B];
	AX_Qty					: ARRAY[1..2] OF UINT	:= [94,			1];
	AX_UnitId				: ARRAY[1..2] OF BYTE	:= [1,			1];
	AX_Function				: ARRAY[1..2] OF UINT	:= [3,			3];	
	AX_Priority				: ARRAY[1..2] OF UINT	:= [1,			1];
END_VAR
// CP-Read / Write 

MesDataExd.MesData.MesCP_Read := MesCP_Read ; 

IF MesCP_Read  THEN	
	

ModbusRTU();
Trig_Read(Clk := CalLocalTimeStruct.wMilliseconds < 200);
IF Trig_Read.Q THEN
	FOR KK := 1 TO 2 DO
			ModbusRTU.M_AddAction_FIFO(InStruct := MbStruct[KK], InPriority := AX_Priority[KK]);
	END_FOR
END_IF

MbStruct[1].InBuffer 	:= ADR(MesBlock_Temp[1]);
MbStruct[1].InFunction 	:= AX_Function[1];
MbStruct[1].InQuantity 	:= AX_Qty[1];
MbStruct[1].InStartAddr := AX_Addr[1];
MbStruct[1].InUnitID 	:= AX_UnitId[1];

MbStruct[2].InBuffer 	:= ADR(MesBlock_Temp[2]);
MbStruct[2].InFunction 	:= AX_Function[2];
MbStruct[2].InQuantity 	:= AX_Qty[2];
MbStruct[2].InStartAddr := AX_Addr[2];
MbStruct[2].InUnitID 	:= AX_UnitId[2];

MW( WORD_STRONG:= MesBlock_Temp[1][0], SIGNED:=FALSE, FIX:=1 , SIZE:=1, VAR_OUT := MesDataExd.MesData.MesI1);
MW( WORD_STRONG:= MesBlock_Temp[1][1], SIGNED:=FALSE, FIX:=1 , SIZE:=1, VAR_OUT := MesDataExd.MesData.MesI2);
MW( WORD_STRONG:= MesBlock_Temp[1][2], SIGNED:=FALSE, FIX:=1 , SIZE:=1, VAR_OUT := MesDataExd.MesData.MesI3);
MW( WORD_STRONG:= MesBlock_Temp[1][4], SIGNED:=FALSE, FIX:=1 , SIZE:=1, VAR_OUT := MesDataExd.MesData.MesI0);
MW( WORD_STRONG:= MesBlock_Temp[1][8], SIGNED:=FALSE, FIX:=1 , SIZE:=1, VAR_OUT := MesDataExd.MesData.MesImax1);
MW( WORD_STRONG:= MesBlock_Temp[1][9], SIGNED:=FALSE, FIX:=1 , SIZE:=1, VAR_OUT := MesDataExd.MesData.MesImax2);
MW( WORD_STRONG:= MesBlock_Temp[1][10], SIGNED:=FALSE, FIX:=1 , SIZE:=1, VAR_OUT := MesDataExd.MesData.MesImax3);
MW( WORD_STRONG:= MesBlock_Temp[1][14], SIGNED:=FALSE, FIX:=0 , SIZE:=1, VAR_OUT := MesDataExd.MesV1);
MW( WORD_STRONG:= MesBlock_Temp[1][15], SIGNED:=FALSE, FIX:=0 , SIZE:=1, VAR_OUT := MesDataExd.MesV2);
MW( WORD_STRONG:= MesBlock_Temp[1][16], SIGNED:=FALSE, FIX:=0 , SIZE:=1, VAR_OUT := MesDataExd.MesV3);
MW( WORD_STRONG:= MesBlock_Temp[1][11], SIGNED:=FALSE, FIX:=0 , SIZE:=1, VAR_OUT := MesDataExd.MesData.MesU12);
MW( WORD_STRONG:= MesBlock_Temp[1][12], SIGNED:=FALSE, FIX:=0 , SIZE:=1, VAR_OUT := MesDataExd.MesData.MesU31);
MW( WORD_STRONG:= MesBlock_Temp[1][13], SIGNED:=FALSE, FIX:=0 , SIZE:=1, VAR_OUT := MesDataExd.MesData.MesU23);
MW( WORD_STRONG:= MesBlock_Temp[1][20], SIGNED:=FALSE, FIX:=2 , SIZE:=1, VAR_OUT := MesDataExd.MesData.MesFreq);
MW( WORD_STRONG:= MesBlock_Temp[1][21], SIGNED:=TRUE, FIX:=0 , SIZE:=1, VAR_OUT := MesDataExd.MesP);
MW( WORD_STRONG:= MesBlock_Temp[1][22], SIGNED:=TRUE, FIX:=0 , SIZE:=1, VAR_OUT := MesDataExd.MesQ);
MW( WORD_STRONG:= MesBlock_Temp[1][23], SIGNED:=TRUE, FIX:=0 , SIZE:=1, VAR_OUT := MesDataExd.MesS);
MW( WORD_STRONG:= MesBlock_Temp[1][26], SIGNED:=TRUE, FIX:=2 , SIZE:=1, VAR_OUT := MesDataExd.MesCosPhi);
MW( WORD_STRONG:= MesBlock_Temp[1][27], WORD_WEAK := MesBlock_Temp[1][28], SIGNED:=FALSE, FIX:=1 , SIZE:=2, VAR_OUT := MesDataExd.EActProd);
MW( WORD_STRONG:= MesBlock_Temp[1][29], WORD_WEAK := MesBlock_Temp[1][30], SIGNED:=FALSE, FIX:=1 , SIZE:=2, VAR_OUT := MesDataExd.EActCons);
MW( WORD_STRONG:= MesBlock_Temp[1][31], WORD_WEAK := MesBlock_Temp[1][32], SIGNED:=FALSE, FIX:=1 , SIZE:=2, VAR_OUT := MesDataExd.EReactProd);
MW( WORD_STRONG:= MesBlock_Temp[1][33], WORD_WEAK := MesBlock_Temp[1][34], SIGNED:=FALSE, FIX:=1 , SIZE:=2, VAR_OUT := MesDataExd.EReactCons);


MesDataExd.Input11 := MesBlock_Temp[2][0].0;
MesDataExd.Input12 := MesBlock_Temp[2][0].1;
MesDataExd.Input13 := MesBlock_Temp[2][0].2;
MesDataExd.Input14 := MesBlock_Temp[2][0].3;
MesDataExd.Input21 := MesBlock_Temp[2][0].4;
MesDataExd.Input22 := MesBlock_Temp[2][0].5;
MesDataExd.Input23 := MesBlock_Temp[2][0].6;
MesDataExd.Input24 := MesBlock_Temp[2][0].7;
MesDataExd.Input25 := MesBlock_Temp[2][0].8;
MesDataExd.Input26 := MesBlock_Temp[2][0].9;

END_IF

// Properties Update 
MesDataExd.MesU := (MesDataExd.MesData.MesU12 + MesDataExd.MesData.MesU31 + MesDataExd.MesData.MesU23 ) /3 ; 

IF MesDataExd.MesP <> 0 THEN
	MesDataExd.MesTanPhi := MesDataExd.MesQ /MesDataExd.MesP;
ELSE
	MesDataExd.MesTanPhi := 0;
END_IF
END_METHOD

END_FUNCTION_BLOCK

// ---- 01_Equipement_Library/Router/FB_Router.TcPOU
FUNCTION_BLOCK FB_Router

VAR_INPUT PERSISTENT 
	ParamTempoRestart		: TIME 		:= T#30S ;	(*  (s)Tempo to wait before resupplying the ADSL routeur*)

	
END_VAR

        	
VAR_INPUT           	
	Heure_Local     		: TIMESTRUCT;
	IN_CmdRestart 			: BOOL;

	
	IN_CmdReset_L			: BOOL ;	// (NA) External Reset Command
	
END_VAR     


VAR_OUTPUT
	//Child objects
	OUT_CmdOpen_IO			: BOOL;	
END_VAR        	
      	
VAR                 	
	bInit					: BOOL;	// Booleen d'initialisation
		
	TP_Restart				: TP;
	// State Mananger //
	MesState				: BYTE; // Cal
	
	// M_Evaluate //	
MesDataExd			: Router_Standard;
END_VAR

METHOD M_AlarmManagement
//////////////////
// Generates object alarms and manages resets. 
//////////////////

VAR 
	// Method local variables (reinitialized at each cycle) 
	FB_AlarmCodeManager		: FB_AlarmCodeManager ;  
END_VAR
	
// ALARM CODE //
	FB_AlarmCodeManager(
		bAlarm1				:= FALSE,						//
		bAlarm2				:= FALSE,                       //
		bAlarm3				:= FALSE,                       //
		bAlarm4				:= FALSE,                       //
		bAlarm5				:= FALSE,                       //
		bAlarm6				:= FALSE,                       //
		bAlarm7				:= FALSE,                       //
		bAlarm8				:= FALSE,                       //
		bAlarm9				:= FALSE,                       //
		bAlarm10			:= FALSE,                       //
		bAlarm11			:= FALSE,                       //
		bAlarm12			:= FALSE,						//
		bAlarm13			:= FALSE ,                      //
		bAlarm14			:= FALSE ,                      //
		bAlarm15			:= FALSE,                       //
		wAlarmCode			=>MesDataExd.MesData.MesAlarmCode);       
			                                                
// WARNING CODE //                                          
	FB_AlarmCodeManager(
		bAlarm1				:= FALSE, 						//				
		bAlarm2				:= FALSE,                       //
		bAlarm3				:= FALSE,                       //
		bAlarm4				:= FALSE,                       //
		bAlarm5				:= FALSE,                       //
		bAlarm6				:= FALSE,                       //
		bAlarm7				:= FALSE,                       //
		bAlarm8				:= FALSE,                       //
		bAlarm9				:= FALSE,                       //
		bAlarm10			:= FALSE,                       //
		bAlarm11			:= FALSE,                       //
		bAlarm12			:= FALSE,                       //
		bAlarm13			:= FALSE,                       //
		bAlarm14			:= FALSE,                       //
		bAlarm15			:= FALSE,                       //
		wAlarmCode			=>MesDataExd.MesData.MesWarningCode);
		
// EVENT CODE //
	FB_AlarmCodeManager(
		bAlarm1			:= OUT_CmdOpen_IO, 					// ADSL is running 
		bAlarm2			:= FALSE , 							//
		bAlarm3			:= FALSE,                           //
		bAlarm4			:= FALSE,                           //
		bAlarm5			:= FALSE,                           //
		bAlarm6			:= FALSE,                           //
		bAlarm7			:= FALSE,                           //
		bAlarm8			:= FALSE,                           //
		bAlarm9			:= FALSE,                           //
		bAlarm10		:= FALSE,                           //
		bAlarm11		:= FALSE,                           //
		bAlarm12		:= FALSE,                           //
		bAlarm13		:= FALSE,                           //
		bAlarm14		:= FALSE,                           //
		bAlarm15		:= FALSE,                           //
		wAlarmCode		=>MesDataExd.MesData.MesEventCode);
END_METHOD

METHOD M_Evaluate
//////////////////
// Evaluate available Powers and AMG characteristics . 
/////////////////

VAR 
	
END_VAR
END_METHOD

METHOD M_Execute : BOOL
VAR_INPUT
END_VAR
IF NOT bInit THEN
	M_Init();
ELSIF CmdClearFault_G OR IN_CmdReset_L THEN
	bInit := TRUE;
ELSE
	
	M_OpenClose(); 
	M_StateManager();
	M_Evaluate();
END_IF
END_METHOD

METHOD M_Init : BOOL
VAR_INPUT
END_VAR
bInit := TRUE;
END_METHOD

METHOD M_OpenClose
//////////////////
// Manages Opening of the contactor
//////////////////

VAR 
	// Method local variables (reinitialized at each cycle) 
	
END_VAR

// Rest Command
TP_Restart(IN:= IN_CmdRestart , PT:=ParamTempoRestart) ;
OUT_CmdOpen_IO	 := TP_Restart.Q ;  // Impulsion that goes back to zero as soon as the state of the TP goes down . 

IF  IN_CmdRestart THEN
	 IN_CmdRestart := FALSE;
END_IF
END_METHOD

METHOD M_StateManager
//////////////////
// Detect which is the state of the inverter. IF loss of communication MesState =0 , the last inverter state is kept .  
/////////////////

VAR 
	// Method local variables (reinitialized at each cycle) 

	
END_VAR
// OPERATIONNAL INDEX //
IF NOT  OUT_CmdOpen_IO THEN 
	MesState.2 := 1;
ELSE
	MesState.0 := 1;
END_IF
END_METHOD

END_FUNCTION_BLOCK

// ---- 01_Equipement_Library/Sensors/ANA/FB_ANA_IO.TcPOU
FUNCTION_BLOCK FB_ANA_IO EXTENDS FB_ANA_Base
//////////////////
// Analogic sensors. Base FB. 
//////////////////

VAR_INPUT PERSISTENT
	// Parameters of the Object (instance/mùodel specific) 
		ParamName				: STRING:='TempPcs';			(* (NA) Name of the pyranometer : to easily identify it *)
		{attribute 'OPC.UA.DA' := '1'}
		ParamScaleMin			: REAL:=4; 						(* (NA) Minimal input value  *)
		{attribute 'OPC.UA.DA' := '1'}
		ParamScaleMax			: REAL:=20; 					(* (NA) Maximal input value  *)
		{attribute 'OPC.UA.DA' := '1'}
		ParamRangeMin			: REAL:=0; 						(* (NA) Minimal output value. Unit depends on output *)
		{attribute 'OPC.UA.DA' := '1'}
		ParamRangeMax			: REAL:=100; 					(* (NA) Maximal output value. Unit depends on output *)

		ParamForced_4_20		: BOOL:=FALSE;				    (* (NA) Is the input between 4-20mA ? *)
		ParamPT100				: BOOL:=FALSE;					(* (NA) PT 100 technology 			  *)
		ParamFix				: INT:=1; 						(* (NA) Value to wich divide the initial value *)
END_VAR

VAR_OUTPUT
	//Child objects
	
END_VAR

VAR_INPUT
    MesDataExd			: ANA_Standard ;     	
	// I/O Inputs 
		//MesIO1				: INT;						 	// 	IO Value
		IN_MesIOReal1			: REAL;
		IN_MesIOReal2			: REAL;
		
END_VAR

VAR
	//M_ALARMMANAGEMENT VARIABLES//
	//M_READ VARIABLES//
		
END_VAR

METHOD M_AlarmManagement
//////////////////
// Manages GHI system alarms and warnings
/////////////////

VAR 
	// Method local variables (reinitialized at each cycle) 

	FB_AlarmCodeManager		: FB_AlarmCodeManager ;   

END_VAR

//RS_MaxAlarm(SET:= MesData.Value > ParamVarMaxAlarm  ,RESET1 := MesData.Value  < (ParamVarMaxAlarm - ParamDiffMax) OR CmdClearFault_G OR IN_CmdReset_L ) ; 

//RS_MaxWarning(SET:=  MesData.Value  > ParamVarMaxWarning  ,RESET1 := MesData.Value  < (ParamVarMaxWarning - ParamDiffMax) OR CmdClearFault_G OR IN_CmdReset_L ) ; 
//RS_MinAlarm(SET:= MesData.Value  < ParamVarMinAlarm  ,RESET1 := MesData.Value  > (ParamVarMinAlarm + ParamDiffMax) OR CmdClearFault_G OR IN_CmdReset_L ) ; 
//RS_MinWarning(SET:=  MesData.Value  < ParamVarMinWarning  ,RESET1 := MesData.Value  > (ParamVarMinWarning + ParamDiffMax) OR CmdClearFault_G OR IN_CmdReset_L ) ; 

RSDiff(SET :=  ABS(MesValue1 - MesValue2) >= ParamDiffMax , RESET1 :=(ABS(MesValue1 - MesValue2) < ParamDiffMax*0.9) OR CmdClearFault_G OR IN_CmdReset_L) ; 


// ALARM CODE //
	FB_AlarmCodeManager(
 		bAlarm1			:= RSDiff.Q1 ,													// The difference between the measured values is higher than 10 %  
		bAlarm2			:= IN_MesVar1Fault_IO OR IN_MesVar2Fault_IO,					// At least one sensor is on fault (0 mA) 
		bAlarm3			:=FALSE , 														// 
		bAlarm4			:=FALSE , 														// 
		bAlarm5			:=FALSE , 														//
		bAlarm6			:=FALSE ,                                                       //
		bAlarm7			:=FALSE ,                                                       //
		bAlarm8			:=FALSE ,                                                       //
		bAlarm9			:=FALSE , 														// 
		bAlarm10		:=FALSE , 														//
		bAlarm11		:=FALSE ,                                                       //
		bAlarm12		:=FALSE ,                                                       //
		bAlarm13		:=FALSE ,                                                       //
		bAlarm14		:=FALSE , 														//
		bAlarm15		:=FALSE ,                                                       //
		wAlarmCode		=>MesDataExd.MesData.MesAlarmCode);                                       
                                                                                        
// WARNING CODE //
	FB_AlarmCodeManager(
		bAlarm1			:= RS_MaxAlarm.Q1,												// Sensor value is higher than Alarm value
		bAlarm2			:= RS_MaxWarning.Q1 ,											// Sensor value is higher than Warning value
		bAlarm3			:= RS_MinAlarm.Q1 ,												// Sensor value is lower than Alarm value 
		bAlarm4			:= RS_MinWarning.Q1 ,											// Sensor value is lower than Warning value 
		bAlarm5			:=FALSE , 														//
		bAlarm6			:=FALSE ,                                       				//
		bAlarm7			:=FALSE ,                                       				//
		bAlarm8			:=FALSE ,                                       				//
		bAlarm9			:=FALSE ,                                       				//
		bAlarm10		:=FALSE ,                                       				//
		bAlarm11		:=FALSE ,                                       				//
		bAlarm12		:=FALSE ,                                       				//
		bAlarm13		:=FALSE ,                                       				//
		bAlarm14		:=FALSE ,                                       				//
		bAlarm15		:=FALSE ,                                       				//
		wAlarmCode		=> MesDataExd.MesData.MesWarningCode);
		
// EVENT CODE //
	FB_AlarmCodeManager(
		bAlarm1			:=FALSE , 														// 
		bAlarm2			:=FALSE , 														// 
		bAlarm3			:=FALSE , 														// 
		bAlarm4			:=FALSE , 														// 
		bAlarm5			:=FALSE , 														//
		bAlarm6			:=FALSE ,       												//
		bAlarm7			:=FALSE ,       												//
		bAlarm8			:=FALSE ,       												//
		bAlarm9			:=FALSE ,       												//
		bAlarm10		:=FALSE ,       												//
		bAlarm11		:=FALSE ,       												//
		bAlarm12		:=FALSE ,       												//
		bAlarm13		:=FALSE ,       												//
		bAlarm14		:=FALSE ,       												//
		bAlarm15		:=FALSE ,       												//
		wAlarmCode		=>MesDataExd.MesData.MesEventCode);
END_METHOD

METHOD M_Read
//////////////////
// Format GHI Data 
/////////////////

VAR 
	// Method local variables (reinitialized at each cycle) 

	
END_VAR
MesValue1 := ((ParamRangeMax - ParamRangeMin) * INT_TO_REAL(IN_MesValue1_IO)/32767)  + ParamRangeMin; 
MesValue2 := ((ParamRangeMax - ParamRangeMin) * INT_TO_REAL(IN_MesValue2_IO)/32767)  + ParamRangeMin; 

IF ParamForced_4_20 THEN
	MesValue1 := ((ParamRangeMax - ParamRangeMin) * ((IN_MesIOReal1 - ParamScaleMin)/(ParamScaleMax-ParamScaleMin)))  + ParamRangeMin; 
	MesValue2 := ((ParamRangeMax - ParamRangeMin) * ((IN_MesIOReal2 - ParamScaleMin)/(ParamScaleMax-ParamScaleMin)))  + ParamRangeMin; 	
END_IF

IF ParamPT100 THEN
	MesValue1	:= INT_TO_REAL(IN_MesValue1_IO) / (EXPT(10,ParamFix)) ; // Param Fix = 1 >> 1/10 , 2 >> 1/100 , 0 >> 1
	MesValue2	:= INT_TO_REAL(IN_MesValue2_IO) / (EXPT(10,ParamFix)) ; // Param Fix = 1 >> 1/10 , 2 >> 1/100 , 0 >> 1	
END_IF

IF ParamNbSensors = 1 THEN 
	MesValue2		:= MesValue1 ;
END_IF

MesDataExd.MesData.Value := (MesValue1  + MesValue2) / 2 ; 			// Mean value ;
END_METHOD

END_FUNCTION_BLOCK

// ---- 01_Equipement_Library/Sensors/ANA/FB_ANA_Base.TcPOU
FUNCTION_BLOCK FB_ANA_Base 
//////////////////
// Analogic sensOR  Base FB. 
//////////////////

VAR_INPUT PERSISTENT
	// Parameters of the Object (instance/mùodel specific) 
	ParamVarMaxAlarm		: REAL 		:=105		; (* (%)  Config : Maximal allowed Site Hygrometry *)
	ParamVarMaxWarning		: REAL 		:=90		; (* (%)  Config : Maximal Site hygrometry warning*)
	ParamVarMinAlarm		: REAL 		:=-5		; (* (%)  Config : Minimal allowed Site Hygrometry *)
	ParamVarMinWarning		: REAL 		:=0			; (* (%)  Config : Minimal Site hygrometry warning*)
	ParamDiffMax			: REAL 		:= 20 		; (* (NA) Config : Maximal Analogic difference acceptable between two sensors*)
	
	ParamNbSensors			: INT 		:=1			; (* (NA) Config : Number of sensors*)
	
END_VAR

VAR_OUTPUT
	//Child objects
	
END_VAR

VAR_INPUT
	// I/O Inputs 
		IN_MesValue1_IO					: UINT ; 		// 	IO Value
		IN_MesValue2_IO					: UINT ; 		// 	IO Value

		IN_MesVar1Fault_IO	AT %I*		: BOOL ; 		//(NA)  sensor 1 has a 0 mA fault  
		IN_MesVar2Fault_IO				: BOOL ; 		//(NA)  sensor 2 has a 0 mA fault  		
END_VAR

VAR
	//M_ALARMMANAGEMENT VARIABLES//

		RS_MaxAlarm: RS;
		RS_MinAlarm: RS;
		RS_MinWarning: RS;
		RS_MaxWarning: RS;
	
		RSDiff: RS;
                                         	
	//M_READ VARIABLES//
		MesValue1						: REAL ;  		// Temporary Value
		MesValue2						: REAL ; 
		
//	MesDataExd					: ANA ; 
			MesCP_Read					: BOOL := TRUE;	(* Read function enable *)
		MesCP_Write					: BOOL := TRUE;	(* Write function enable *)
		
		// M_INIT //
		bInit 							: BOOL;
		IN_CmdReset_L					: BOOL;
END_VAR

METHOD M_AlarmManagement
//////////////////
// Manages GHI system alarms and warnings
/////////////////

VAR 
	// Method local variables (reinitialized at each cycle) 
 	FB_AlarmCodeManager		: FB_AlarmCodeManager ; 
	

END_VAR
END_METHOD

METHOD M_Execute
//////////////////
//  Method Calls 
/////////////////

VAR 
	// Method local variables (reinitialized at each cycle) 

END_VAR
// METHODS CALLS // 
	M_Read(); 
	M_AlarmManagement() ;
END_METHOD

METHOD M_Read
//////////////////
// Format GHI Data 
/////////////////

VAR 
	// Method local variables (reinitialized at each cycle) 
END_VAR
END_METHOD

END_FUNCTION_BLOCK

// ---- 01_Equipement_Library/Sensors/ANA/FB_ANA_Irra_Fx.TcPOU
FUNCTION_BLOCK FB_ANA_Irra_Fx EXTENDS FB_ANA_Base
//////////////////
// (4-20 mA) sensor . 
//////////////////

VAR_INPUT PERSISTENT
	// Parameters of the Object (instance/model specific) 
	ParamSensibility				: REAL:=1 ;		(* (mV/W.m2) Pyranometer sensibility. Scale often : -200 W/m2 >> 0 mV , 2000 W/m2 >> 32 mV*) 
	ParamFactorConvertisseur		: REAL := 10 ; (* (mA/mV) Coefficient de conversion mV en mA. Default value = 2  *)
		{attribute 'OPC.UA.DA' := '1'}
		ParamScaleMin			: REAL:=4; 						(* (NA) Minimal input value  *)
		{attribute 'OPC.UA.DA' := '1'}
		ParamScaleMax			: REAL:=20; 					(* (NA) Maximal input value  *)
		{attribute 'OPC.UA.DA' := '1'}
		ParamRangeMin			: REAL:=0; 						(* (NA) Minimal output value. Unit depends on output *)
		{attribute 'OPC.UA.DA' := '1'}
		ParamRangeMax			: REAL:=1600; 					(* (NA) Maximal output value. Unit depends on output *)
	
	
	
END_VAR

VAR_OUTPUT
	//Child objects
	
END_VAR

VAR_INPUT
	// I/O Inputs 
	IN_MesReal1_IO			: UINT;
END_VAR         			
                			
VAR    


    MesData					: ANA ;     

         			
	A						: REAL;     // F(x) = Ax+B
	B						: REAL;     // F(x) = Ax+B


		
END_VAR

METHOD M_AlarmManagement
//////////////////
// Manages GHI system alarms and warnings
/////////////////

VAR 
	// Method local variables (reinitialized at each cycle) 

	FB_AlarmCodeManager		: FB_AlarmCodeManager ;   

END_VAR

RS_MaxAlarm(SET:= MesData.Value > ParamVarMaxAlarm  ,RESET1 := MesData.Value  < (ParamVarMaxAlarm - ParamDiffMax) OR CmdClearFault_G OR IN_CmdReset_L ) ; 

RS_MaxWarning(SET:=  MesData.Value  > ParamVarMaxWarning  ,RESET1 := MesData.Value  < (ParamVarMaxWarning - ParamDiffMax) OR CmdClearFault_G OR IN_CmdReset_L ) ; 
RS_MinAlarm(SET:= MesData.Value  < ParamVarMinAlarm  ,RESET1 := MesData.Value  > (ParamVarMinAlarm + ParamDiffMax) OR CmdClearFault_G OR IN_CmdReset_L ) ; 
RS_MinWarning(SET:=  MesData.Value  < ParamVarMinWarning  ,RESET1 := MesData.Value  > (ParamVarMinWarning + ParamDiffMax) OR CmdClearFault_G OR IN_CmdReset_L ) ; 

RSDiff(SET :=  ABS(MesValue1 - MesValue2) >= ParamDiffMax , RESET1 :=(ABS(MesValue1 - MesValue2) < ParamDiffMax*0.9) OR CmdClearFault_G OR IN_CmdReset_L) ; 


// ALARM CODE //
	FB_AlarmCodeManager(
 		bAlarm1			:= RSDiff.Q1 ,													// The difference between the measured values is higher than 10 %  
		bAlarm2			:= IN_MesVar1Fault_IO OR IN_MesVar2Fault_IO,					// At least one sensor is on fault (0 mA) 
		bAlarm3			:=FALSE , 														// 
		bAlarm4			:=FALSE , 														// 
		bAlarm5			:=FALSE , 														//
		bAlarm6			:=FALSE ,                                                       //
		bAlarm7			:=FALSE ,                                                       //
		bAlarm8			:=FALSE ,                                                       //
		bAlarm9			:=FALSE , 														// 
		bAlarm10		:=FALSE , 														//
		bAlarm11		:=FALSE ,                                                       //
		bAlarm12		:=FALSE ,                                                       //
		bAlarm13		:=FALSE ,                                                       //
		bAlarm14		:=FALSE , 														//
		bAlarm15		:=FALSE ,                                                       //
		wAlarmCode		=>MesData.MesAlarmCode);                                       
                                                                                        
// WARNING CODE //
	FB_AlarmCodeManager(
		bAlarm1			:= RS_MaxAlarm.Q1,												// Sensor value is higher than Alarm value
		bAlarm2			:= RS_MaxWarning.Q1 ,											// Sensor value is higher than Warning value
		bAlarm3			:= RS_MinAlarm.Q1 ,												// Sensor value is lower than Alarm value 
		bAlarm4			:= RS_MinWarning.Q1 ,											// Sensor value is lower than Warning value 
		bAlarm5			:=FALSE , 														//
		bAlarm6			:=FALSE ,                                       				//
		bAlarm7			:=FALSE ,                                       				//
		bAlarm8			:=FALSE ,                                       				//
		bAlarm9			:=FALSE ,                                       				//
		bAlarm10		:=FALSE ,                                       				//
		bAlarm11		:=FALSE ,                                       				//
		bAlarm12		:=FALSE ,                                       				//
		bAlarm13		:=FALSE ,                                       				//
		bAlarm14		:=FALSE ,                                       				//
		bAlarm15		:=FALSE ,                                       				//
		wAlarmCode		=>MesData.MesWarningCode);
		
// EVENT CODE //
	FB_AlarmCodeManager(
		bAlarm1			:=FALSE , 														// 
		bAlarm2			:=FALSE , 														// 
		bAlarm3			:=FALSE , 														// 
		bAlarm4			:=FALSE , 														// 
		bAlarm5			:=FALSE , 														//
		bAlarm6			:=FALSE ,       												//
		bAlarm7			:=FALSE ,       												//
		bAlarm8			:=FALSE ,       												//
		bAlarm9			:=FALSE ,       												//
		bAlarm10		:=FALSE ,       												//
		bAlarm11		:=FALSE ,       												//
		bAlarm12		:=FALSE ,       												//
		bAlarm13		:=FALSE ,       												//
		bAlarm14		:=FALSE ,       												//
		bAlarm15		:=FALSE ,       												//
		wAlarmCode		=>MesData.MesEventCode);
END_METHOD

METHOD M_Read
//////////////////
// Format GHI Data 
/////////////////

VAR 
	// Method local variables (reinitialized at each cycle) 
	MesValue_420mA : REAL;
	MesValue_mV	: REAL ; 
END_VAR
(*	IF ParamSensibility > 0.1	THEN  
		A := (ParamRangeMax-ParamRangeMin)/(ParamScaleMax-ParamScaleMin)*ParamFactorConvertisseur / ParamSensibility; 
		B :=  (ParamRangeMin*ParamScaleMax -ParamRangeMax*ParamScaleMin)/(ParamScaleMax-ParamScaleMin) * ParamFactorConvertisseur / ParamSensibility;
	ELSE
		A:=0 ; 
		B:=0 ; 
	END_IF
*)
	
	// Convert 0 >> 32767 to 4-20 mA . 
	MesValue_420mA := ((ParamScaleMax-ParamScaleMin)/(32767-0)*(IN_MesReal1_IO-0))+ParamScaleMin;		// 
	
	// Convert in mV 
	MesValue_mV		:= (MesValue_420mA - ParamScaleMin) * ParamFactorConvertisseur ; 	// Consider that mV starts at 0  . 
	
	// Convert in W /m2 et mise à l'echelle
	MesData.Value := SEL( ABS(ParamSensibility)< 0.01 ,   MesValue_mV / ParamSensibility , 0 ) ; // Does not take in account voltage offset . 
	
	// Convert 4-20 mA to 0 >> 1600 W/m2 
	
	
	//MesData.Value := A*MesValue_420mA + B;
END_METHOD

END_FUNCTION_BLOCK

// ---- 01_Equipement_Library/Sensors/COM/FB_AllInOne.TcPOU
FUNCTION_BLOCK FB_AllInOne
VAR_INPUT
	ParamNameAllInOne		: STRING 	:= 'Wind spd + dir + hygro + temp';				// (NA) Name of the pyranometer : to easily identify it
	ParamTempoComAlarm		: TIME 		:= T#10S ; 										// (s) Config : Tempo to detect LOC Alarm
	{attribute 'OPC.UA.DA' := '1'} 
	ParamClockReadTime 		: TIME 		:= T#2S;	  									// (Time) Read Modbus Frequency . 
 	ParamTimeout			: TIME  	:= T#5S ;		  								// (Time) Timeout for modbus reading
	{attribute 'OPC.UA.DA' := '1'} 
	ParamUnitID				: BYTE		:= 1;											// (NA) Unit ID for modbus reading
	{attribute 'OPC.UA.DA' := '1'} 
	ParamTCPPort			: UINT		:= 502;											// (NA) TCP port for modbus
	{attribute 'OPC.UA.DA' := '1'} 
	ParamIpAddress			: STRING	:= '127.0.0.1';									// (NA) IP address for modbus
END_VAR

VAR
	//M_AlarmManagement
	TON_ComAlarm				: TON ; 								// Tempo before deteting loss of communication. 

	
	IN_CmdReset_L					: BOOL;                                                        	
		
	// M_READ VARIABLES//
MesData		AT %Q*  : AllInOne ; 							// (NA) [P,H,B] INV  Data Structure 
	FB_ModbusReadInputRegs		: ARRAY[1..2] OF FB_MBReadInputRegs;	// FB for Modbus Read
	MesBlock1_Temp 				: ARRAY[1..96]  OF WORD; 				// (NA) Temporary Block with multiple modbus reading (Caution : Double Word variables)
	MesBlock2_Temp 				: ARRAY[1..3]  OF WORD; 				// (NA) Temporary Block with multiple modbus reading (Caution : Double Word variables)
	MesModbusReadAlarm1 		: BOOL ; 								// (NA) Modbus Read Alarm for all modbus frames		
	MesModbusReadAlarm2 		: BOOL ; 								// (NA) Modbus Read Alarm for all modbus frames		
	MesAlarmCom					: BOOL;                         		
	MesModbusAlarmCode			: UDINT;								// (NA) Modbus Read Alarm Code	
	                                                            		
	// M_STATEMANAGER//                                         		
	FB_OperationIndex			: FB_OperationIndex ;           		
	MesLastStart				: STRING ;			 					// Datetime of the last Start
	MesState					: BYTE ; 								// (NA) Cal                                                                                                            	
	MesRunningTime				: INT ; 								// Total Running Time
	                                                        			
	//M_EXECUTE VARIABLES //                                		
	TP1							: TP ; 									// (NA) Tempo to define Modbus Reading Frequency 
	                                                        	
	ClockRead				AT %Q*	: BOOL;								// (NA) Modbus reading Clock
	
	
	//M_INIT //
	bInit 						: BOOL;							 
END_VAR

VAR_OUTPUT
END_VAR
VAR
END_VAR

METHOD M_AlarmManagement
//////////////////
// Manages IntelliGen Alarms
/////////////////

VAR 
	// Method local variables (reinitialized at each cycle) 
	FB_AlarmCodeManager : FB_AlarmCodeManager ; 
END_VAR

TON_ComAlarm(IN:= (MesModbusReadAlarm1) AND (MesModbusReadAlarm2) , PT:= ParamTempoComAlarm, Q=>MesAlarmCom) ;	

FB_AlarmCodeManager(
		bAlarm1			:= MesAlarmCom,  					// No connexion to inverter 
		bAlarm2			:= FALSE,//
		bAlarm3			:= False,//
		bAlarm4			:= False,//
		bAlarm5			:= False,//
		bAlarm6			:= FALSE, 							//
		bAlarm7			:= False, 							//
		bAlarm8			:= False, 							//
		bAlarm9			:= False, 							//
		bAlarm10		:= False, 							//
		bAlarm11		:= FALSE,                         //
		bAlarm12		:= FALSE,                         //
		bAlarm13		:= FALSE,                         //
		bAlarm14		:= FALSE, 							// 
		bAlarm15		:= FALSE , 			// 
		wAlarmCode		=>MesData.MesAlarmCode);
END_METHOD

METHOD M_Execute
//////////////////
//  Method Calls 
/////////////////

VAR 
	// Method local variables (reinitialized at each cycle) 

END_VAR
IF NOT bInit THEN
	M_Init();
END_IF

// READING AND WRITING CLOCK //
	TP1(IN:=NOT TP1.Q , PT:= ParamClockReadTime);
	ClockRead 				:= TP1.Q;
	
	

// METHODS CALLS//
	M_Read();



	/////////
	M_StateManager() ; 
	

	M_AlarmManagement();
END_METHOD

METHOD M_Init : BOOL
VAR_INPUT
END_VAR


bInit := FALSE;
END_METHOD

{attribute 'object_name' := 'M_Read'}
METHOD M_Read
//////////
// Read Method for SMA : Modbus reading
//////////
VAR
	// Method local variables (reinitialized at each cycle) 
	MW 					: FB_MergeWordsToDint; 
	tets : uint;
END_VAR

FB_ModbusReadInputRegs[1]
(	
	pDestAddr := ADR(MesBlock1_Temp),
	sIPAddr := ParamIpAddress,
	tTimeout := T#1S,
	nQuantity := 96,
	ntcpport := ParamTCPPort,
	nMBAddr := 0,
	cbLength := 96*2,
	nUnitID := 1,
	bExecute := ClockRead,
	nErrId => MesModbusAlarmCode,
	bError => MesModbusReadAlarm1
);
FB_ModbusReadInputRegs[2]
(	
	pDestAddr := ADR(MesBlock2_Temp),
	sIPAddr := ParamIpAddress,
	tTimeout := T#1S,
	nQuantity := 3,
	ntcpport := ParamTCPPort,
	nMBAddr := 4128,
	cbLength := 3*2,
	nUnitID := 1,
	bExecute := ClockRead,
	nErrId => MesModbusAlarmCode,
	bError => MesModbusReadAlarm2
);
	


	
MW(WORD_STRONG := MesBlock1_Temp[65], size := 1, fix := 1,SIGNED := TRUE, VAR_OUT := MesData.MesTemp_Amb);
MW(WORD_STRONG := MesBlock1_Temp[66], size := 1, fix := 0,SIGNED := FALSE, VAR_OUT := MesData.MesAlarmTemp);
MW(WORD_STRONG := MesBlock1_Temp[3], size := 1, fix := 1,SIGNED := TRUE, VAR_OUT := MesData.MesHygro);
MW(WORD_STRONG := MesBlock1_Temp[4], size := 1, fix := 0,SIGNED := FALSE, VAR_OUT := MesData.MesAlarmHygro);
MW(WORD_STRONG := MesBlock1_Temp[5], size := 1, fix := 1,SIGNED := TRUE, VAR_OUT := MesData.MesDewPoint);
MW(WORD_STRONG := MesBlock1_Temp[6], size := 1, fix := 0,SIGNED := FALSE, VAR_OUT := MesData.MesAlarmDewPt);
MW(WORD_STRONG := MesBlock1_Temp[93], size := 1, fix := 2,SIGNED := TRUE, VAR_OUT := MesData.MesWindSp);
MW(WORD_STRONG := MesBlock1_Temp[94], size := 1, fix := 0,SIGNED := FALSE, VAR_OUT := MesData.MesAlarmWindSp);
MW(WORD_STRONG := MesBlock1_Temp[95], size := 1, fix := 1,SIGNED := TRUE, VAR_OUT := MesData.MesWindDir);
MW(WORD_STRONG := MesBlock1_Temp[96], size := 1, fix := 0,SIGNED := FALSE, VAR_OUT := MesData.MesAlarmWindDir);

	
MW(WORD_STRONG := MesBlock2_Temp[1], size := 1, fix := 0,SIGNED := TRUE, VAR_OUT := MesData.MesRain1);
MW(WORD_STRONG := MesBlock2_Temp[2], size := 1, fix := 0,SIGNED := TRUE, VAR_OUT := MesData.MesRain2);
MW(WORD_STRONG := MesBlock2_Temp[3], size := 1, fix := 0,SIGNED := TRUE, VAR_OUT := MesData.MesRain3);
END_METHOD

METHOD M_StateManager
//////////////////
// Detect which is the state of the inverter. IF loss of communication MesState =0 , the last inverter state is kept .  
/////////////////

VAR 
	// Method local variables (reinitialized at each cycle) 

	
END_VAR
// OPERATIONNAL INDEX //
//	FB_OperationIndex(
//		MesON 				:= MesState>1, 
//		CmdReset 			:= CmdReInitMaintenanceIndicator_G,
//		CalRunningTimeHr 	=> CalRunningTime , 
//		CalNbMove 			=> CalNbMove,
//		CalTimeStart 		=> CalLastStart) ;
END_METHOD

END_FUNCTION_BLOCK

// ---- 01_Equipement_Library/Sensors/COM/FB_ANA_SMP1X.TcPOU
FUNCTION_BLOCK FB_ANA_SMP1X
VAR_INPUT PERSISTENT
	
	ParamNamePyranometer	: STRING 	:= 'Wind spd + dir + hygro + temp + pluvio';	// (NA) Name of the eqt : to easily identify it
	ParamTempoComAlarm		: TIME 		:= T#10S ; 										// (s) Config : Tempo to detect LOC Alarm
	{attribute 'OPC.UA.DA' := '1'} 
	ParamClockReadTime 		: TIME 		:= TIME#1S;	  									// (Time) Read Modbus Frequency . 
 	ParamTimeout			: TIME  	:= T#2S ;		  								// (Time) Timeout for modbus reading
	ParamUnitID				: BYTE		:= 1;											// (NA) Unit ID for modbus reading
	ParamZonePTR			: BOOL;														// (NA) Is the Pyranometer connected on the PTR
END_VAR

VAR_INPUT
	MesDataExd			    : SMP1X ; 					// (NA) [P,H,B] INV  Data Structure 
	IN_CmdToggleRead		: BOOL;
	
END_VAR
VAR
	//M_AlarmManagement
	TON_ComAlarm				: TON ; 						// Tempo before deteting loss of communication. 

	MesAlarmCom					: BOOL;
	
	IN_CmdReset_L					: BOOL;                                                        	

	
	// M_READ VARIABLES//
		MesData	AT %Q*	      	: SMP1X ; 					// (NA) [P,H,B] INV  Data Structure 
	//ModbusRead_RTU				: FB_ReadModbusRTU_V2;			// FB for Modbus Read
	bReadError					: BOOL;
	bReadCompleted 				: BOOL;
	bReadBusy					: BOOL;
	ReadErrorId					: INT;
	InputStructRead 			: Struct_InputRTU;
	
	MesBlock1_Temp 				: ARRAY[1..125]  OF WORD; 		// (NA) Temporary Block with multiple modbus reading (Caution : Double Word variables)
	MesModbusReadAlarm 		  	: BOOL ; 						// (NA) Modbus Read Alarm for all modbus frames		
	MesModbusAlarmCode			: UDINT;						// (NA) Modbus Read Alarm Code	
	
	ScaleFactor					: REAL;
	BodyTemp					: REAL;
	StatusFlag					: REAL;
	
	// M_STATEMANAGER//
	FB_OperationIndex			: FB_OperationIndex ; 
	CalLastStart				: STRING ;			 			// Datetime of the last Start
	MesState					: BYTE ; 						// (NA)                                                                                                            	
	CalRunningTime				: INT ; 						// Total Running Time
	                                                        	
	//M_EXECUTE VARIABLES //                                	
	TP1							: TP ; 							// (NA) Tempo to define Modbus Reading Frequency 
	                                                        	
	ClockRead					: BOOL;							// (NA) Modbus reading Clock
	Trig_ClockRead				: R_TRIG;
	Trig_Cmd_Read : R_TRIG;
	
	//M_INIT //
	bInit 						: BOOL;							 
END_VAR

VAR_OUTPUT
END_VAR
VAR
END_VAR

METHOD M_AlarmManagement
//////////////////
// Manages IntelliGen Alarms
/////////////////

VAR 
	// Method local variables (reinitialized at each cycle) 
	FB_AlarmCodeManager : FB_AlarmCodeManager ; 
	ComWarning			: BOOL;		// Aggregated Wcommunication warning
	ComAlarm			: BOOL;		// Aggregated communication Alarm

END_VAR
 
		
		ComAlarm	:=  MesModbusReadAlarm;

	//Warning
	
	//Alarm
	TON_ComAlarm(IN:= ComAlarm , PT:= ParamTempoComAlarm, Q=>MesAlarmCom) ;	// Alarms if ALL TRAM MODBUS did not work and timeout of 15s


// ALARM CODE //
	FB_AlarmCodeManager(
		bAlarm1			:= MesAlarmCom,  						// Com alarm
		bAlarm2			:= MesDataExd.MesAlarm = 1 , 								
		bAlarm3			:= MesDataExd.MesAlarm = 2 , 										 
		bAlarm4			:= FALSE,      							
		bAlarm5			:= FALSE,								
		bAlarm6			:= FALSE,								
		bAlarm7			:= FALSE,                               
		bAlarm8			:= FALSE,                               
		bAlarm9			:= FALSE,								
		bAlarm10		:= FALSE,					            
		bAlarm11		:= FALSE,                               
		bAlarm12		:= FALSE,                               
		bAlarm13		:= FALSE,                               
		bAlarm14		:= FALSE, 								
		bAlarm15		:= FALSE , 								
		wAlarmCode		=>MesDataExd.MesData.MesAlarmCode);     

// WARNING CODE //
	FB_AlarmCodeManager(
 		bAlarm1			:= FALSE ,				
		bAlarm2			:= FALSE,				
		bAlarm3			:= FALSE,				
		bAlarm4			:= FALSE, 				
		bAlarm5			:= FALSE,				
		bAlarm6			:= FALSE,				
		bAlarm7			:= FALSE, 
		bAlarm8			:= FALSE, 
		bAlarm9			:= FALSE, 
		bAlarm10		:= FALSE, 
		bAlarm11		:= FALSE, 
		bAlarm12		:= FALSE, 
		bAlarm13		:= FALSE, 
		bAlarm14		:= FALSE, 
		bAlarm15		:= FALSE, 
		wAlarmCode		=>MesDataExd.MesData.MesWarningCode);
END_METHOD

METHOD M_CP : BOOL
VAR_INPUT
END_VAR
END_METHOD

METHOD M_Execute
//////////////////
//  Method Calls 
/////////////////

VAR 
	// Method local variables (reinitialized at each cycle) 

END_VAR
IF NOT bInit THEN
	M_Init();
ELSIF GVL_CFG.CmdClearFault_G OR IN_CmdReset_L THEN
	bInit := TRUE;
END_IF

// READING AND WRITING CLOCK //
	TP1(IN:=NOT TP1.Q , PT:= ParamClockReadTime);
	ClockRead 				:= TP1.Q;
	
	

// METHODS CALLS//
	M_CP();
	
	M_Read();


	/////////
	M_StateManager() ; 
	

	M_AlarmManagement();
END_METHOD

METHOD M_Init : BOOL
VAR_INPUT
END_VAR


bInit := FALSE;
END_METHOD

{attribute 'object_name' := 'M_Read'}
METHOD M_Read
//////////
// Read Method for SMA : Modbus reading
//////////
VAR
	// Method local variables (reinitialized at each cycle) 
	MW 					: FB_MergeWordsToDint; 
	
	Val_Interm: REAL;
END_VAR
InputStructRead.InBuffer := ADR(MesBlock1_Temp);
InputStructRead.InFunction := 4;
InputStructRead.InQuantity := 8;
InputStructRead.InStartAddr := 3;
InputStructRead.InUnitID := ParamUnitID;
InputStructRead.OutBusy := ADR(bReadBusy);
InputStructRead.OutError := ADR(bReadError);
InputStructRead.OutCompleted := ADR(bReadCompleted);



IF MesDataExd.MesCP_Read THEN
	MW(WORD_STRONG := MesBlock1_Temp[1], SIZE:= 1, Fix := 0, SIGNED := FALSE, VAR_OUT := StatusFlag);
	MW(WORD_STRONG := MesBlock1_Temp[2], SIZE:= 1, Fix := 0, SIGNED := FALSE, VAR_OUT := ScaleFactor);
	MW(WORD_STRONG := MesBlock1_Temp[3], SIZE:= 1, Fix := 0, SIGNED := FALSE, VAR_OUT := MesDataExd.MesData.Value);
END_IF
MesDataExd.MesAlarm := StatusFlag;
END_METHOD

METHOD M_StateManager
//////////////////
// Detect which is the state of the inverter. IF loss of communication MesState =0 , the last inverter state is kept .  
/////////////////

VAR 
	// Method local variables (reinitialized at each cycle) 

	
END_VAR
// OPERATIONNAL INDEX //
//	FB_OperationIndex(
//		MesON 				:= MesState>1, 
//		CmdReset 			:= CmdReInitMaintenanceIndicator_G,
//		CalRunningTimeHr 	=> CalRunningTime , 
//		CalNbMove 			=> CalNbMove,
//		CalTimeStart 		=> CalLastStart) ;
END_METHOD

END_FUNCTION_BLOCK

// ---- 01_Equipement_Library/Sensors/TOR/FB_TOR_CB.TcPOU
FUNCTION_BLOCK FB_TOR_CB EXTENDS FB_TOR_Base
//////////////////
//  Circuit Breaker
//////////////////

VAR_INPUT PERSISTENT
	// Parameters of the Object (instance/model specific) 
	ParamTP_Impulsion		    : TIME 		:= T#2S;	(* (s) Config : Tempo for the start or stop command impulsion*)
	ParamNC_Tripped				: BOOL;		(* (NA) is the tripped signal normally closed: True = Normally closed*)
		
END_VAR

VAR_OUTPUT
	//Child objects
	OUT_CmdOpen_IO	           : BOOL ; 	          // (NA) Physical I/O Open Command IO
	OUT_CmdClose_IO			   : BOOL ; 	          // (NA) Physical I/O Close Command IO
	
END_VAR

VAR_INPUT
	// I/O Inputs 		                                     				
		IN_CmdOpen 						: BOOL ; 				// (NA) External Open Command 
		IN_CmdClose						: BOOL ; 				// (NA) External Close Command 
		IN_MesTripped_IO				: BOOL ;				// (NA) the CB tripped
		
END_VAR

VAR
	//M_ALARMMANAGEMENT VARIABLES//
		
		MesDataExd			: TOR_CB ;  

	//M_OPENCLOSE VARIABLES//	
		ParamTP_Open	 			: TP ;				(* (NA) Temporisation for Open pulse Command*)
		ParamTP_Close 				: TP ;				(* (NA) Temporisation for Close pulse Command	*)

END_VAR

METHOD M_AlarmManagement
//////////////////
// Manages Door sensor alarms and warnings
/////////////////

VAR 
	// Method local variables (reinitialized at each cycle) 
	FB_AlarmCodeManager : FB_AlarmCodeManager ; 


END_VAR
IF ParamNC_Tripped THEN
	MesDataExd.MesTripped := NOT IN_MesTripped_IO;
ELSE
	MesDataExd.MesTripped := IN_MesTripped_IO;
END_IF

// ALARM CODE //
	FB_AlarmCodeManager(
 		bAlarm1			:= MesDataExd.MesTripped,    					// 
		bAlarm2			:= FALSE, 						// 
		bAlarm3			:= FALSE, 						// 
		bAlarm4			:= FALSE, 						// 
		bAlarm5			:= FALSE,       				//
		bAlarm6			:= FALSE,       				//
		bAlarm7			:= FALSE,       				//
		bAlarm8			:= FALSE,       				//
		bAlarm9			:= FALSE,       				//
		bAlarm10		:= FALSE,       				//
		bAlarm11		:= FALSE,       				//
		bAlarm12		:= FALSE,         				//
		bAlarm13		:= FALSE,         				//
		bAlarm14		:= FALSE,         				//
		bAlarm15		:= FALSE,         				//
		wAlarmCode		=>MesDataExd.MesData.MesAlarmCode);

// WARNING CODE //
	FB_AlarmCodeManager(
		bAlarm1			:= FALSE,    			// 
		bAlarm2			:= FALSE, 				//  
		bAlarm3			:= FALSE, 				//  
		bAlarm4			:= FALSE, 				//  
		bAlarm5			:= FALSE,               //
		bAlarm6			:= FALSE,               //
		bAlarm7			:= FALSE,               //
		bAlarm8			:= FALSE,               //
		bAlarm9			:= FALSE,               //
		bAlarm10		:= FALSE,               //
		bAlarm11		:= FALSE,               //
		bAlarm12		:= FALSE,               //
		bAlarm13		:= FALSE,               //
		bAlarm14		:= FALSE,               //
		bAlarm15		:= FALSE,               //
		wAlarmCode		=>MesDataExd.MesData.MesWarningCode);

// EVENT CODE //
	FB_AlarmCodeManager(
		bAlarm1			:= MesDataExd.MesData.MesAlarmState, 			//  CB is opened
		bAlarm2			:= FALSE, 							// 
		bAlarm3			:= FALSE, 							//  
		bAlarm4			:= FALSE, 							// 
		bAlarm5			:= FALSE,                           //
		bAlarm6			:= FALSE,                           //
		bAlarm7			:= FALSE,                           //
		bAlarm8			:= FALSE,                           //
		bAlarm9			:= FALSE,                           //
		bAlarm10		:= FALSE,                           //
		bAlarm11		:= FALSE,                           //
		bAlarm12		:= FALSE,                           //
		bAlarm13		:= FALSE,                           //
		bAlarm14		:= FALSE,                           //
		bAlarm15		:= FALSE,                           //
		wAlarmCode		=>MesDataExd.MesData.MesEventCode);
END_METHOD

METHOD M_StateManager
//////////////////
// Detect when fire occurs
/////////////////

VAR 
	// Method local variables (reinitialized at each cycle)
 	MesStateInterm1 : BOOL;
	MesStateInterm2 : BOOL;
END_VAR

IF ParamCableCutSecurity THEN
	MesStateInterm1 := NOT IN_MesState1_IO ; 
	MesStateInterm2 := NOT IN_MesState2_IO ; 
ELSE 
	MesStateInterm1 := IN_MesState1_IO;
	MesStateInterm2 := IN_MesState2_IO;
END_IF

IF ParamNbSensors = 1 THEN 
	MesStateInterm2 := MesStateInterm1 ;
END_IF

IF ParamAtleastOne THEN 
	MesDataExd.MesData.MesAlarmState := MesStateInterm1 OR MesStateInterm2 ; 
ELSE
	MesDataExd.MesData.MesAlarmState := MesStateInterm1 AND MesStateInterm2 ; 
END_IF

R_TRIGAlarm(CLK:= MesDataExd.MesData.MesAlarmState ) ; 
IF R_TRIGAlarm.Q THEN
	MesCountAlarm :=  MIN(MesCountAlarm + 1 ,4294967295 ) ; 
ELSIF IN_ResetCounter THEN 
	MesCountAlarm := 0 ; 
END_IF

MesDataExd.MesData.MesCountAlarm	:= MesCountAlarm ; 

MesDataExd.MesCP_Open				:= IN_CmdOpen AND NOT IN_CmdReset_L;
MesDataExd.MesCP_Close				:= MesDataExd.MesData.MesAlarmState AND IN_CmdClose AND NOT MesDataExd.MesData.MesAlarmCode.0 AND NOT MesDataExd.MesCP_Open AND NOT IN_CmdReset_L ;
// Open Command
ParamTP_Open(IN		:= MesDataExd.MesCP_Open , PT:=ParamTP_Impulsion) ;
OUT_CmdOpen_IO		:= ParamTP_Open.Q ;                               			 // Impulsion that goes back to zero as soon as the state of the TP goes down. 

// Close Command
ParamTP_Close(IN	:= MesDataExd.MesCP_Close , PT:=ParamTP_Impulsion) ;
OUT_CmdClose_IO		:= ParamTP_Close.Q ;                          				 // Impulsion that goes back to zero as soon as the state of the TP goes down.
END_METHOD

END_FUNCTION_BLOCK

// ---- 01_Equipement_Library/Sensors/TOR/FB_TOR_Base.TcPOU
FUNCTION_BLOCK FB_TOR_Base
//////////////////
//  Digital SensOR  Base FB . 
//////////////////

VAR_INPUT PERSISTENT
	// Parameters of the Object (instance/model specific) 
	ParamNbSensors					: INT 		:=1		; 	(* (NA) Config : Number of sensors, If =9 Then sensor is bi-stable contactor*)
	ParamAtleastOne					: BOOL 		:= TRUE ;  	(* (NA) If TRUE, the output is true if at leat one of the sensor is active. Otherwise, the output is true only if both are active*)
	ParamCableCutSecurity			: BOOL		:=FALSE;	(* (NA) FALSE = ALARM *)
	                        		
	MesCountAlarm					: UDINT 	:=0 ; 		// (NA) Cal : Count number of times the alarm has been triggered
	
END_VAR

VAR_OUTPUT
	//Child objects
	
END_VAR

VAR_INPUT
	// I/O Inputs 		                                     				
		IN_MesState1_IO 			: BOOL ;	 		// (NA) First  Smoke detector IO, IF bi-stable NC
		IN_MesState2_IO				: BOOL ; 			// (NA) Second Smoke detector IO, IF Bi-stable NO
		IN_CmdReset_L				: BOOL ;			// LOCAL Reset Value For Alarms
		IN_ResetCounter 			: BOOL ; 			// Reset counter
END_VAR

VAR
	//M_ALARMMANAGEMENT VARIABLES//

	//STATE MANAGEMENT //
//	MesDataExd				: TOR ; 	
		R_TRIGAlarm					: R_TRIG ; 

			MesCP_Read					: BOOL := TRUE;	(* Read function enable *)
		MesCP_Write					: BOOL := TRUE;	(* Write function enable *)
	
END_VAR

METHOD M_AlarmManagement
//////////////////
// Manages Door sensor alarms and warnings
/////////////////

VAR 
	// Method local variables (reinitialized at each cycle) 


END_VAR
END_METHOD

METHOD M_Execute
//////////////////
//  Method Calls 
/////////////////

VAR 
	// Method local variables (reinitialized at each cycle) 
	
END_VAR
// METHODS CALLS // 
	M_StateManager() ; // order is important 
	M_AlarmManagement() ;
END_METHOD

METHOD M_StateManager
//////////////////
// Detect when fire occurs
/////////////////

VAR 
	// Method local variables (reinitialized at each cycle)
 	MesStateInterm1 : BOOL;
	MesStateInterm2 : BOOL;
END_VAR
END_METHOD

END_FUNCTION_BLOCK

// ---- 01_Equipement_Library/Sensors/TOR/FB_TOR_Standard.TcPOU
FUNCTION_BLOCK FB_TOR_Standard EXTENDS FB_TOR_Base
//////////////////
//  Circuit Breaker
//////////////////

VAR_INPUT PERSISTENT
	// Parameters of the Object (instance/model specific) 
		
		
END_VAR

VAR_OUTPUT
	//Child objects
	
END_VAR

VAR_INPUT
	// I/O Inputs 		                                     				
		
END_VAR

VAR
	//M_ALARMMANAGEMENT VARIABLES//
		
MesDataExd			: TOR_Standard ;  

	
END_VAR

METHOD M_AlarmManagement
//////////////////
// Manages Door sensor alarms and warnings
/////////////////

VAR 
	// Method local variables (reinitialized at each cycle) 
	FB_AlarmCodeManager : FB_AlarmCodeManager ; 


END_VAR

// ALARM CODE //
	FB_AlarmCodeManager(
 		bAlarm1			:= FALSE,    					// 
		bAlarm2			:= FALSE, 						// 
		bAlarm3			:= FALSE, 						// 
		bAlarm4			:= FALSE, 						// 
		bAlarm5			:= FALSE,       				//
		bAlarm6			:= FALSE,       				//
		bAlarm7			:= FALSE,       				//
		bAlarm8			:= FALSE,       				//
		bAlarm9			:= FALSE,       				//
		bAlarm10		:= FALSE,       				//
		bAlarm11		:= FALSE,       				//
		bAlarm12		:= FALSE,         				//
		bAlarm13		:= FALSE,         				//
		bAlarm14		:= FALSE,         				//
		bAlarm15		:= FALSE,         				//
		wAlarmCode		=>MesDataExd.MesData.MesAlarmCode);

// WARNING CODE //
	FB_AlarmCodeManager(
		bAlarm1			:= FALSE,    			// 
		bAlarm2			:= FALSE, 				//  
		bAlarm3			:= FALSE, 				//  
		bAlarm4			:= FALSE, 				//  
		bAlarm5			:= FALSE,               //
		bAlarm6			:= FALSE,               //
		bAlarm7			:= FALSE,               //
		bAlarm8			:= FALSE,               //
		bAlarm9			:= FALSE,               //
		bAlarm10		:= FALSE,               //
		bAlarm11		:= FALSE,               //
		bAlarm12		:= FALSE,               //
		bAlarm13		:= FALSE,               //
		bAlarm14		:= FALSE,               //
		bAlarm15		:= FALSE,               //
		wAlarmCode		=>MesDataExd.MesData.MesWarningCode);

// EVENT CODE //
	FB_AlarmCodeManager(
		bAlarm1			:= MesDataExd.MesData.MesAlarmState, 			//  CB is opened
		bAlarm2			:= FALSE, 							// 
		bAlarm3			:= FALSE, 							//  
		bAlarm4			:= FALSE, 							// 
		bAlarm5			:= FALSE,                           //
		bAlarm6			:= FALSE,                           //
		bAlarm7			:= FALSE,                           //
		bAlarm8			:= FALSE,                           //
		bAlarm9			:= FALSE,                           //
		bAlarm10		:= FALSE,                           //
		bAlarm11		:= FALSE,                           //
		bAlarm12		:= FALSE,                           //
		bAlarm13		:= FALSE,                           //
		bAlarm14		:= FALSE,                           //
		bAlarm15		:= FALSE,                           //
		wAlarmCode		=>MesDataExd.MesData.MesEventCode);
END_METHOD

METHOD M_StateManager
//////////////////
// Detect when fire occurs
/////////////////

VAR 
	// Method local variables (reinitialized at each cycle)
 	MesStateInterm1 : BOOL;
	MesStateInterm2 : BOOL;
END_VAR

IF ParamCableCutSecurity THEN
	MesStateInterm1 := NOT IN_MesState1_IO ; 
	MesStateInterm2 := NOT IN_MesState2_IO ; 
ELSE 
	MesStateInterm1 := IN_MesState1_IO;
	MesStateInterm2 := IN_MesState2_IO;
END_IF

IF ParamNbSensors = 1 THEN 
	MesStateInterm2 := MesStateInterm1 ;
END_IF

IF ParamAtleastOne THEN 
MesDataExd.MesData.MesAlarmState := MesStateInterm1 OR MesStateInterm2 ; 
ELSE
MesDataExd.MesData.MesAlarmState := MesStateInterm1 AND MesStateInterm2 ; 
END_IF

R_TRIGAlarm(CLK:= MesDataExd.MesData.MesAlarmState ) ; 
IF R_TRIGAlarm.Q THEN
	MesCountAlarm :=  MIN(MesCountAlarm + 1 ,4294967295 ) ; 
ELSIF IN_ResetCounter THEN 
	MesCountAlarm := 0 ; 
END_IF

MesDataExd.MesData.MesCountAlarm	:= MesCountAlarm ;
END_METHOD

END_FUNCTION_BLOCK

// ---- 01_Equipement_Library/Sensors/TOR/FB_TOR_ES.TcPOU
FUNCTION_BLOCK FB_TOR_ES EXTENDS FB_TOR_Base
//////////////////
//  Emergency stop system
//////////////////
VAR_INPUT PERSISTENT
	// Parameters of the Object (instance/model specific) 
	ParamTempoEs :TIME:=T#2S;								(* (s) Tempo before raising an alarm*)
END_VAR

VAR_OUTPUT
	//Child objects
	
END_VAR

VAR_INPUT
	// I/O Inputs 		                                     				
		
	
END_VAR

VAR
	//M_ALARMMANAGEMENT VARIABLES//
		FB_PermAlarm				: SR ;					// (NA) FB to maintain emergency stop Alarm 
		TON_ES						: TON ; 
 
	//M_STATEMANAGER VARIABLES//
		MesDataExd			: TOR_Standard ;  	
END_VAR

METHOD M_AlarmManagement
//////////////////
// Manages Smoke detector alarms and warnings
/////////////////

VAR 
	// Method local variables (reinitialized at each cycle) 
	FB_AlarmCodeManager			: FB_AlarmCodeManager ; 
	bAlarmsNbSensors			: BOOL;
END_VAR
// Detection Variables
TON_ES(IN:= MesDataExd.MesData.MesAlarmState , PT:= ParamTempoEs ); 
FB_PermAlarm(SET1 := TON_ES.Q, Reset := CmdClearFault_G OR IN_CmdReset_L); 							// SR FB for keep fire if burn

bAlarmsNbSensors	:= SEL(ParamNbSensors=9,FALSE, IN_MesState1_IO <> IN_MesState2_IO);
// ALARM CODE //
	FB_AlarmCodeManager(
		bAlarm1			:= FB_PermAlarm.Q1,  														// Emergency stop		
		bAlarm2			:= bAlarmsNbSensors, 														// Incoherent measures between sensors
		bAlarm3			:=FALSE, 																	// 
		bAlarm4			:=FALSE, 																	// 
		bAlarm5			:=FALSE, 																	//
		bAlarm6			:=FALSE,                                                                    //
		bAlarm7			:=FALSE,                                                                    //
		bAlarm8			:=FALSE,                                                                    //
		bAlarm9			:=FALSE,                                                                    //
		bAlarm10		:=FALSE,                                                                    //
		bAlarm11		:=FALSE,                                                                    //
		bAlarm12		:=FALSE,                                                                    //
		bAlarm13		:=FALSE,                                                                    //
		bAlarm14		:=FALSE,                                                                    //
		bAlarm15		:=FALSE,                                                                    //
		wAlarmCode		=>MesDataExd.MesData.MesAlarmCode );
		
// WARNING CODE //
	FB_AlarmCodeManager(
		bAlarm1			:=IN_MesState1_IO OR IN_MesState2_IO,	 	 								// At least one detector is ON 
		bAlarm2			:=FALSE, 																	// 
		bAlarm3			:=FALSE, 																	// 
		bAlarm4			:=FALSE, 																	// 
		bAlarm5			:=FALSE, 																	//
		bAlarm6			:=FALSE,                                                                    //
		bAlarm7			:=FALSE,                                                                    //
		bAlarm8			:=FALSE,                                                                    //
		bAlarm9			:=FALSE,                                                                    //
		bAlarm10		:=FALSE,                                                                    //
		bAlarm11		:=FALSE,                                                                    //
		bAlarm12		:=FALSE,                                                                    //
		bAlarm13		:=FALSE,                                                                    //
		bAlarm14		:=FALSE,                                                                    //
		bAlarm15		:=FALSE,                                                                    //
		wAlarmCode		=>MesDataExd.MesData.MesWarningCode);
		
// EVENT CODE //
	FB_AlarmCodeManager(
		bAlarm1			:= IN_MesState1_IO, 														// First sensor is ON
		bAlarm2			:= IN_MesState2_IO, 														// Second sensor is ON
		bAlarm3			:= FALSE, 																	// 
		bAlarm4			:= FALSE, 																	// 
		bAlarm5			:= FALSE, 																	//
		bAlarm6			:= FALSE,                   												//
		bAlarm7			:= FALSE,                   												//
		bAlarm8			:= FALSE,                   												//
		bAlarm9			:= FALSE,                   												//
		bAlarm10		:= FALSE,                   												//
		bAlarm11		:= FALSE,                   												//
		bAlarm12		:= FALSE,                   												//
		bAlarm13		:= FALSE,                   												//
		bAlarm14		:= FALSE,                   												//
		bAlarm15		:= FALSE,                   												//
		wAlarmCode		=>MesDataExd.MesData.MesEventCode);
END_METHOD

METHOD M_Execute
//////////////////
//  Method Calls 
/////////////////

VAR 
	// Method local variables (reinitialized at each cycle) 

END_VAR

	
	IF ParamNbSensors = 9 THEN // Use of contactor bi-stable No and NC
		IN_MesState2_IO := NOT IN_MesState2_IO;
	END_IF
SUPER^.M_Execute() ;
END_METHOD

METHOD M_StateManager
//////////////////
// Detect when fire occurs
/////////////////

VAR 
	// Method local variables (reinitialized at each cycle)
 	MesStateInterm1 : BOOL;
	MesStateInterm2 : BOOL;
END_VAR

IF ParamCableCutSecurity THEN
	MesStateInterm1 := NOT IN_MesState1_IO ; 
	MesStateInterm2 := NOT IN_MesState2_IO ; 
ELSE 
	MesStateInterm1 := IN_MesState1_IO;
	MesStateInterm2 := IN_MesState2_IO;
END_IF

IF ParamNbSensors = 1 THEN 
	MesStateInterm2 :=  MesStateInterm1;
END_IF

IF ParamAtleastOne THEN 
MesDataExd.MesData.MesAlarmState := MesStateInterm1 OR MesStateInterm2 ; 
ELSE
MesDataExd.MesData.MesAlarmState := MesStateInterm1 AND MesStateInterm2 ; 
END_IF

R_TRIGAlarm(CLK:= MesDataExd.MesData.MesAlarmState ) ; 
IF R_TRIGAlarm.Q THEN
	MesCountAlarm :=  MIN(MesCountAlarm + 1 ,4294967295 ) ; 
ELSIF IN_ResetCounter THEN 
	MesCountAlarm := 0 ; 
END_IF

MesDataExd.MesData.MesCountAlarm	:= MesCountAlarm ;
END_METHOD

END_FUNCTION_BLOCK

// ---- 01_Equipement_Library/Sensors/TOR/FB_TOR_Fuse.TcPOU
FUNCTION_BLOCK FB_TOR_Fuse EXTENDS FB_TOR_Base
//////////////////
//  Smoke and Fire detection system with Typhoon triggering system. 
//////////////////
VAR_INPUT PERSISTENT
	// Parameters of the Object (instance/model specific) 
	ParamTempoFuse :TIME:=T#5S;//  (s)Tempo before raising an alarm
END_VAR

VAR_OUTPUT
	//Child objects
	
END_VAR

VAR_INPUT
	// I/O Inputs 		                                     				
		
	
END_VAR

VAR
	//M_ALARMMANAGEMENT VARIABLES//
		FB_PermAlarm				: SR ;					// (NA) FB to maintain Fire Alarm even if sensor stop detection (burn) .
 		TON_Fuse					: TON; 	
	//M_STATEMANAGER VARIABLES//
	MesDataExd			: TOR_Standard ;  

		
END_VAR

METHOD M_AlarmManagement
//////////////////
// Manages Smoke detector alarms and warnings
/////////////////

VAR 
	// Method local variables (reinitialized at each cycle) 
	FB_AlarmCodeManager			: FB_AlarmCodeManager ; 

	bAlarmsNbSensors: BOOL;
END_VAR
// Detection Variables
TON_Fuse(IN:= MesDataExd.MesData.MesAlarmState , PT:= ParamTempoFuse ) ; 
FB_PermAlarm(SET1 := TON_Fuse.Q  , Reset := CmdClearFault_G OR IN_CmdReset_L ); // SR FB for keep fire if burn .

bAlarmsNbSensors	:= SEL(ParamNbSensors=9,FALSE, IN_MesState1_IO <> IN_MesState2_IO);
// ALARM CODE //
	FB_AlarmCodeManager(
		bAlarm1			:= FB_PermAlarm.Q1 ,  														// Fuse is burned 		
		bAlarm2			:= bAlarmsNbSensors, 														// Incoherent measures between sensors
		bAlarm3			:=FALSE, 																	// 
		bAlarm4			:=FALSE, 																	// 
		bAlarm5			:=FALSE, 																	//
		bAlarm6			:=FALSE,                                                                    //
		bAlarm7			:=FALSE,                                                                    //
		bAlarm8			:=FALSE,                                                                    //
		bAlarm9			:=FALSE,                                                                    //
		bAlarm10		:=FALSE,                                                                    //
		bAlarm11		:=FALSE,                                                                    //
		bAlarm12		:=FALSE,                                                                    //
		bAlarm13		:=FALSE,                                                                    //
		bAlarm14		:=FALSE,                                                                    //
		bAlarm15		:=FALSE,                                                                    //
		wAlarmCode		=>MesDataExd.MesData.MesAlarmCode );
		
// WARNING CODE //
	FB_AlarmCodeManager(
		bAlarm1			:= IN_MesState1_IO OR  IN_MesState2_IO,	  								// At least one sensor is on.  
		bAlarm2			:=FALSE, 																// 
		bAlarm3			:=FALSE, 																// 
		bAlarm4			:=FALSE, 																// 
		bAlarm5			:=FALSE, 																//
		bAlarm6			:=FALSE,                                                                //
		bAlarm7			:=FALSE,                                                                //
		bAlarm8			:=FALSE,                                                                //
		bAlarm9			:=FALSE,                                                                //
		bAlarm10		:=FALSE,                                                                //
		bAlarm11		:=FALSE,                                                                //
		bAlarm12		:=FALSE,                                                                //
		bAlarm13		:=FALSE,                                                                //
		bAlarm14		:=FALSE,                                                                //
		bAlarm15		:=FALSE,                                                                //
		wAlarmCode			=>MesDataExd.MesData.MesWarningCode);
		
// EVENT CODE //
	FB_AlarmCodeManager(
		bAlarm1			:= IN_MesState1_IO, 													// First sensor is ON
		bAlarm2			:= IN_MesState2_IO, 													// Second sensor is ON
		bAlarm3			:= FALSE, 																// 
		bAlarm4			:= FALSE, 																// 
		bAlarm5			:= FALSE, 																//
		bAlarm6			:= FALSE,                                                               //
		bAlarm7			:= FALSE,                                                               //
		bAlarm8			:= FALSE,                                                               //
		bAlarm9			:= FALSE,                                                               //
		bAlarm10		:= FALSE,                                                               //
		bAlarm11		:= FALSE,                                                               //
		bAlarm12		:= FALSE,                                                               //
		bAlarm13		:= FALSE,                                                               //
		bAlarm14		:= FALSE,                                                               //
		bAlarm15		:= FALSE,                                                               //
		wAlarmCode		=>MesDataExd.MesData.MesEventCode);
END_METHOD

METHOD M_Execute
//////////////////
//  Method Calls 
/////////////////

VAR 
	// Method local variables (reinitialized at each cycle) 

END_VAR
// EMULATOR I/O //

	
	IF ParamNbSensors = 9 THEN // Use of contactor bi-stable No and NC
		IN_MesState2_IO := NOT IN_MesState2_IO;
	END_IF
SUPER^.M_Execute() ;
END_METHOD

METHOD M_StateManager
//////////////////
// Detect when fire occurs
/////////////////

VAR 
	// Method local variables (reinitialized at each cycle)
 	MesStateInterm1 : BOOL;
	MesStateInterm2 : BOOL;
END_VAR

IF ParamCableCutSecurity THEN
	MesStateInterm1 := NOT IN_MesState1_IO ; 
	MesStateInterm2 := NOT IN_MesState2_IO ; 
ELSE 
	MesStateInterm1 := IN_MesState1_IO;
	MesStateInterm2 := IN_MesState2_IO;
END_IF

IF ParamNbSensors = 1 THEN 
	MesStateInterm2 := MesStateInterm1 ;
END_IF

IF ParamAtleastOne THEN 
MesDataExd.MesData.MesAlarmState := MesStateInterm1 OR MesStateInterm2 ; 
ELSE
MesDataExd.MesData.MesAlarmState := MesStateInterm1 AND MesStateInterm2 ; 
END_IF

R_TRIGAlarm(CLK:= MesDataExd.MesData.MesAlarmState ) ; 
IF R_TRIGAlarm.Q THEN
	MesCountAlarm :=  MIN(MesCountAlarm + 1 ,4294967295 ) ; 
ELSIF IN_ResetCounter THEN 
	MesCountAlarm := 0 ; 
END_IF

MesDataExd.MesData.MesCountAlarm	:= MesCountAlarm ;
END_METHOD

END_FUNCTION_BLOCK

// ---- 01_Equipement_Library/Sensors/TOR/FB_TOR_MS.TcPOU
FUNCTION_BLOCK FB_TOR_MS EXTENDS FB_TOR_Base
//////////////////
//  Motion Sensor System
//////////////////

VAR_INPUT PERSISTENT
	// Parameters of the Object (instance/model specific) 
		ParamTempoDoorAlarm			: TIME := T#10S ;	(* (S) Tempo for Door sensor alarm *)
		ParamTempoUnlockAlarm		: TIME := T#1800S ;	(* (S) Tempo for Door sensor alarm *)
END_VAR

VAR_OUTPUT
	//Child objects
	
END_VAR

VAR_INPUT
	// I/O Inputs 		                                     				
		
END_VAR

VAR
	//M_ALARMMANAGEMENT VARIABLES//
	
		TON_Fermeture			: TON;				//(NA) Tempo to detect door opened for too long time . 
		PT_Unlock_Alarm			: TP;				//(NA) Timer to unlock alarm after 30 min
		
		MesDataExd			: TOR_Standard ;  

END_VAR

METHOD M_AlarmManagement
//////////////////
// Manages Door sensor alarms and warnings
/////////////////

VAR 
	// Method local variables (reinitialized at each cycle) 
	FB_AlarmCodeManager : FB_AlarmCodeManager ; 

END_VAR
// Detection Variables

// The Motion Sensor must be activated for the duration of ParamTempoDoorAlarm for the alarm to be activated
TON_Fermeture(IN:= MesDataExd.MesData.MesAlarmState,PT:=ParamTempoDoorAlarm); //

// ALARM CODE //
	FB_AlarmCodeManager(
 		bAlarm1			:= FALSE,    							// 
		bAlarm2			:= FALSE, 								// 
		bAlarm3			:= FALSE, 								// 
		bAlarm4			:= FALSE, 								// 
		bAlarm5			:= FALSE,    							// 
		bAlarm6			:= FALSE, 								// 
		bAlarm7			:= FALSE, 								// 
		bAlarm8			:= FALSE, 								// 
		bAlarm9			:= FALSE,    							// 
		bAlarm10		:= FALSE, 								// 
		bAlarm11		:= FALSE, 								// 
		bAlarm12		:= FALSE, 								// 
		bAlarm13		:= FALSE,								// 
		bAlarm14		:= FALSE,								// 
		bAlarm15		:= FALSE,								// 
		wAlarmCode		=>MesDataExd.MesData.MesAlarmCode);

